LIN {X 0,Y 573.245,Z 183.073,A -85,B 0,C 180,E1 -2299.475,E2 -2299.475} C_VEL
LIN {X 0,Y 573.228,Z 183.082,A -85,B 0,C 180,E1 -2302.192,E2 -2302.192} C_VEL
LIN {X 0,Y 573.232,Z 183.075,A -85,B 0,C 180,E1 -2305.229,E2 -2305.229} C_VEL
LIN {X 0,Y 573.246,Z 183.076,A -85,B 0,C 180,E1 -2307.773,E2 -2307.773} C_VEL
LIN {X 0,Y 573.242,Z 183.077,A -85,B 0,C 180,E1 -2310.633,E2 -2310.633} C_VEL
LIN {X 0,Y 573.208,Z 183.078,A -85,B 0,C 180,E1 -2313.022,E2 -2313.022} C_VEL
LIN {X 0,Y 573.235,Z 183.076,A -85,B 0,C 180,E1 -2315.364,E2 -2315.364} C_VEL
LIN {X 0,Y 573.23,Z 183.08,A -85,B 0,C 180,E1 -2317.662,E2 -2317.662} C_VEL
LIN {X 0,Y 573.266,Z 183.072,A -85,B 0,C 180,E1 -2320.67,E2 -2320.67} C_VEL
LIN {X 0,Y 573.23,Z 183.082,A -85,B 0,C 180,E1 -2323.621,E2 -2323.621} C_VEL
LIN {X 0,Y 573.258,Z 183.081,A -85,B 0,C 180,E1 -2325.807,E2 -2325.807} C_VEL
LIN {X 0,Y 573.264,Z 183.071,A -85,B 0,C 180,E1 -2328.745,E2 -2328.745} C_VEL
LIN {X 0,Y 573.282,Z 183.078,A -85,B 0,C 180,E1 -2331.54,E2 -2331.54} C_VEL
LIN {X 0,Y 573.289,Z 183.068,A -85,B 0,C 180,E1 -2334.372,E2 -2334.372} C_VEL
LIN {X 0,Y 573.317,Z 183.067,A -85,B 0,C 180,E1 -2337.892,E2 -2337.892} C_VEL
LIN {X 0,Y 573.322,Z 183.066,A -85,B 0,C 180,E1 -2340.702,E2 -2340.702} C_VEL
LIN {X 0,Y 573.297,Z 183.071,A -85,B 0,C 180,E1 -2342.811,E2 -2342.811} C_VEL
LIN {X 0,Y 573.299,Z 183.071,A -85,B 0,C 180,E1 -2345.628,E2 -2345.628} C_VEL
LIN {X 0,Y 573.254,Z 183.074,A -85,B 0,C 180,E1 -2348.46,E2 -2348.46} C_VEL
LIN {X 0,Y 573.273,Z 183.077,A -85,B 0,C 180,E1 -2351.312,E2 -2351.312} C_VEL
LIN {X 0,Y 573.282,Z 183.073,A -85,B 0,C 180,E1 -2354.424,E2 -2354.424} C_VEL
LIN {X 0,Y 573.258,Z 183.079,A -85,B 0,C 180,E1 -2357.112,E2 -2357.112} C_VEL
LIN {X 0,Y 573.241,Z 183.076,A -85,B 0,C 180,E1 -2360.077,E2 -2360.077} C_VEL
LIN {X 0,Y 573.241,Z 183.118,A -85,B 0,C 180,E1 -2362.1,E2 -2362.1} C_VEL
LIN {X 0,Y 573.215,Z 193.051,A -85,B 0,C 180,E1 -2364.168,E2 -2364.168} C_VEL
LIN {X 0,Y 572.806,Z 194.29,A -85,B 0,C 180,E1 -2364.24,E2 -2364.24} C_VEL
LIN {X 0,Y 570.997,Z 198.736,A -85,B 0,C 180,E1 -2364.254,E2 -2364.254} C_VEL
LIN {X 0,Y 568.332,Z 207.365,A -85,B 0,C 180,E1 -2364.283,E2 -2364.283} C_VEL
LIN {X 0,Y 567.483,Z 212.853,A -85,B 0,C 180,E1 -2364.307,E2 -2364.307} C_VEL
LIN {X 0,Y 567.099,Z 223.962,A -85,B 0,C 180,E1 -2364.48,E2 -2364.48} C_VEL
LIN {X 0,Y 566.981,Z 298.738,A -85,B 0,C 180,E1 -2365.445,E2 -2365.445} C_VEL
LIN {X 0,Y 566.829,Z 311.548,A -85,B 0,C 180,E1 -2365.744,E2 -2365.744} C_VEL
LIN {X 0,Y 566.743,Z 323.735,A -85,B 0,C 180,E1 -2366.168,E2 -2366.168} C_VEL
LIN {X 0,Y 566.592,Z 335.861,A -85,B 0,C 180,E1 -2366.737,E2 -2366.737} C_VEL
LIN {X 0,Y 566.431,Z 347.166,A -85,B 0,C 180,E1 -2367.428,E2 -2367.428} C_VEL
LIN {X 0,Y 566.322,Z 357.588,A -85,B 0,C 180,E1 -2368.225,E2 -2368.225} C_VEL
LIN {X 0,Y 566.2,Z 367.478,A -85,B 0,C 180,E1 -2369.156,E2 -2369.156} C_VEL
LIN {X 0,Y 566.096,Z 376.256,A -85,B 0,C 180,E1 -2370.186,E2 -2370.186} C_VEL
LIN {X 0,Y 566.001,Z 383.39,A -85,B 0,C 180,E1 -2371.215,E2 -2371.215} C_VEL
LIN {X 0,Y 565.948,Z 389.91,A -85,B 0,C 180,E1 -2372.389,E2 -2372.389} C_VEL
LIN {X 0,Y 565.92,Z 395.392,A -85,B 0,C 180,E1 -2373.69,E2 -2373.69} C_VEL
LIN {X 0,Y 565.869,Z 399.185,A -85,B 0,C 180,E1 -2374.945,E2 -2374.945} C_VEL
LIN {X 0,Y 565.822,Z 401.595,A -85,B 0,C 180,E1 -2376.162,E2 -2376.162} C_VEL
LIN {X 0,Y 565.831,Z 402.879,A -85,B 0,C 180,E1 -2377.489,E2 -2377.489} C_VEL
LIN {X 0,Y 565.817,Z 402.903,A -85,B 0,C 180,E1 -2378.508,E2 -2378.508} C_VEL
LIN {X 0,Y 565.851,Z 401.989,A -85,B 0,C 180,E1 -2379.641,E2 -2379.641} C_VEL
LIN {X 0,Y 565.841,Z 400.12,A -85,B 0,C 180,E1 -2380.743,E2 -2380.743} C_VEL
LIN {X 0,Y 565.925,Z 396.386,A -85,B 0,C 180,E1 -2382.114,E2 -2382.114} C_VEL
LIN {X 0,Y 565.95,Z 392.76,A -85,B 0,C 180,E1 -2383.078,E2 -2383.078} C_VEL
LIN {X 0,Y 565.98,Z 386.895,A -85,B 0,C 180,E1 -2384.279,E2 -2384.279} C_VEL
LIN {X 0,Y 566.059,Z 379.21,A -85,B 0,C 180,E1 -2385.506,E2 -2385.506} C_VEL
LIN {X 0,Y 566.158,Z 371.385,A -85,B 0,C 180,E1 -2386.504,E2 -2386.504} C_VEL
LIN {X 0,Y 566.222,Z 362.446,A -85,B 0,C 180,E1 -2387.433,E2 -2387.433} C_VEL
LIN {X 0,Y 566.39,Z 352.66,A -85,B 0,C 180,E1 -2388.263,E2 -2388.263} C_VEL
LIN {X 0,Y 566.483,Z 340.994,A -85,B 0,C 180,E1 -2389.062,E2 -2389.062} C_VEL
LIN {X 0,Y 566.666,Z 329.627,A -85,B 0,C 180,E1 -2389.666,E2 -2389.666} C_VEL
LIN {X 0,Y 566.81,Z 317.931,A -85,B 0,C 180,E1 -2390.142,E2 -2390.142} C_VEL
LIN {X 0,Y 566.897,Z 304.866,A -85,B 0,C 180,E1 -2390.521,E2 -2390.521} C_VEL
LIN {X 0,Y 567.002,Z 292.327,A -85,B 0,C 180,E1 -2390.742,E2 -2390.742} C_VEL
LIN {X 0,Y 567.076,Z 198.669,A -85,B 0,C 180,E1 -2391.934,E2 -2391.934} C_VEL
LIN {X 0,Y 566.144,Z 193.381,A -85,B 0,C 180,E1 -2392.029,E2 -2392.029} C_VEL
LIN {X 0,Y 566.23,Z 183.952,A -85,B 0,C 180,E1 -2394.046,E2 -2394.046} C_VEL
LIN {X 0,Y 566.2,Z 183.956,A -85,B 0,C 180,E1 -2396.897,E2 -2396.897} C_VEL
LIN {X 0,Y 566.172,Z 183.962,A -85,B 0,C 180,E1 -2399.407,E2 -2399.407} C_VEL
LIN {X 0,Y 566.194,Z 183.953,A -85,B 0,C 180,E1 -2401.857,E2 -2401.857} C_VEL
LIN {X 0,Y 566.194,Z 183.952,A -85,B 0,C 180,E1 -2404.25,E2 -2404.25} C_VEL
LIN {X 0,Y 566.171,Z 183.959,A -85,B 0,C 180,E1 -2407.368,E2 -2407.368} C_VEL
LIN {X 0,Y 566.204,Z 183.952,A -85,B 0,C 180,E1 -2409.663,E2 -2409.663} C_VEL
LIN {X 0,Y 566.182,Z 183.953,A -85,B 0,C 180,E1 -2411.921,E2 -2411.921} C_VEL
LIN {X 0,Y 566.192,Z 183.953,A -85,B 0,C 180,E1 -2414.153,E2 -2414.153} C_VEL
LIN {X 0,Y 566.186,Z 183.956,A -85,B 0,C 180,E1 -2416.359,E2 -2416.359} C_VEL
LIN {X 0,Y 566.237,Z 183.955,A -85,B 0,C 180,E1 -2418.676,E2 -2418.676} C_VEL
LIN {X 0,Y 566.204,Z 183.951,A -85,B 0,C 180,E1 -2421.434,E2 -2421.434} C_VEL
LIN {X 0,Y 566.263,Z 183.948,A -85,B 0,C 180,E1 -2424.302,E2 -2424.302} C_VEL
LIN {X 0,Y 566.283,Z 183.942,A -85,B 0,C 180,E1 -2427.866,E2 -2427.866} C_VEL
LIN {X 0,Y 566.299,Z 183.945,A -85,B 0,C 180,E1 -2430.711,E2 -2430.711} C_VEL
LIN {X 0,Y 566.26,Z 183.947,A -85,B 0,C 180,E1 -2432.846,E2 -2432.846} C_VEL
LIN {X 0,Y 566.253,Z 183.946,A -85,B 0,C 180,E1 -2435.699,E2 -2435.699} C_VEL
LIN {X 0,Y 566.224,Z 183.954,A -85,B 0,C 180,E1 -2438.566,E2 -2438.566} C_VEL
LIN {X 0,Y 566.244,Z 183.946,A -85,B 0,C 180,E1 -2441.454,E2 -2441.454} C_VEL
LIN {X 0,Y 566.225,Z 183.952,A -85,B 0,C 180,E1 -2444.502,E2 -2444.502} C_VEL
LIN {X 0,Y 566.189,Z 183.953,A -85,B 0,C 180,E1 -2447.332,E2 -2447.332} C_VEL
LIN {X 0,Y 566.202,Z 183.954,A -85,B 0,C 180,E1 -2449.581,E2 -2449.581} C_VEL
LIN {X 0,Y 566.188,Z 183.96,A -85,B 0,C 180,E1 -2451.863,E2 -2451.863} C_VEL
LIN {X 0,Y 566.184,Z 183.953,A -85,B 0,C 180,E1 -2455.022,E2 -2455.022} C_VEL
LIN {X 0,Y 566.173,Z 183.957,A -85,B 0,C 180,E1 -2457.341,E2 -2457.341} C_VEL
LIN {X 0,Y 566.173,Z 183.964,A -85,B 0,C 180,E1 -2459.771,E2 -2459.771} C_VEL
LIN {X 0,Y 566.202,Z 183.952,A -85,B 0,C 180,E1 -2462.429,E2 -2462.429} C_VEL
LIN {X 0,Y 566.179,Z 183.955,A -85,B 0,C 180,E1 -2464.989,E2 -2464.989} C_VEL
LIN {X 0,Y 566.193,Z 183.959,A -85,B 0,C 180,E1 -2467.461,E2 -2467.461} C_VEL
LIN {X 0,Y 566.208,Z 183.951,A -85,B 0,C 180,E1 -2470.199,E2 -2470.199} C_VEL
LIN {X 0,Y 566.195,Z 183.955,A -85,B 0,C 180,E1 -2473.055,E2 -2473.055} C_VEL
LIN {X 0,Y 566.161,Z 183.957,A -85,B 0,C 180,E1 -2476.053,E2 -2476.053} C_VEL
LIN {X 0,Y 566.168,Z 183.958,A -85,B 0,C 180,E1 -2478.86,E2 -2478.86} C_VEL
LIN {X 0,Y 566.207,Z 183.957,A -85,B 0,C 180,E1 -2481.443,E2 -2481.443} C_VEL
LIN {X 0,Y 566.152,Z 183.957,A -85,B 0,C 180,E1 -2484.307,E2 -2484.307} C_VEL
LIN {X 0,Y 566.198,Z 183.957,A -85,B 0,C 180,E1 -2486.896,E2 -2486.896} C_VEL
LIN {X 0,Y 566.171,Z 183.96,A -85,B 0,C 180,E1 -2489.407,E2 -2489.407} C_VEL
LIN {X 0,Y 566.155,Z 183.957,A -85,B 0,C 180,E1 -2491.854,E2 -2491.854} C_VEL
LIN {X 0,Y 566.203,Z 183.951,A -85,B 0,C 180,E1 -2494.25,E2 -2494.25} C_VEL
LIN {X 0,Y 566.165,Z 183.958,A -85,B 0,C 180,E1 -2497.368,E2 -2497.368} C_VEL
LIN {X 0,Y 566.203,Z 183.951,A -85,B 0,C 180,E1 -2499.662,E2 -2499.662} C_VEL
LIN {X 0,Y 566.177,Z 183.954,A -85,B 0,C 180,E1 -2501.921,E2 -2501.921} C_VEL
LIN {X 0,Y 566.185,Z 183.955,A -85,B 0,C 180,E1 -2504.152,E2 -2504.152} C_VEL
LIN {X 0,Y 566.172,Z 183.959,A -85,B 0,C 180,E1 -2506.358,E2 -2506.358} C_VEL
LIN {X 0,Y 566.234,Z 183.948,A -85,B 0,C 180,E1 -2509.27,E2 -2509.27} C_VEL
LIN {X 0,Y 566.22,Z 183.952,A -85,B 0,C 180,E1 -2512.153,E2 -2512.153} C_VEL
LIN {X 0,Y 566.261,Z 183.946,A -85,B 0,C 180,E1 -2515.016,E2 -2515.016} C_VEL
LIN {X 0,Y 566.282,Z 183.943,A -85,B 0,C 180,E1 -2517.866,E2 -2517.866} C_VEL
LIN {X 0,Y 566.294,Z 183.944,A -85,B 0,C 180,E1 -2520.711,E2 -2520.711} C_VEL
LIN {X 0,Y 566.252,Z 183.947,A -85,B 0,C 180,E1 -2522.846,E2 -2522.846} C_VEL
LIN {X 0,Y 566.249,Z 183.947,A -85,B 0,C 180,E1 -2525.698,E2 -2525.698} C_VEL
LIN {X 0,Y 566.201,Z 183.955,A -85,B 0,C 180,E1 -2528.566,E2 -2528.566} C_VEL
LIN {X 0,Y 566.243,Z 183.947,A -85,B 0,C 180,E1 -2531.454,E2 -2531.454} C_VEL
LIN {X 0,Y 566.228,Z 183.95,A -85,B 0,C 180,E1 -2534.502,E2 -2534.502} C_VEL
LIN {X 0,Y 566.163,Z 183.957,A -85,B 0,C 180,E1 -2537.333,E2 -2537.333} C_VEL
LIN {X 0,Y 566.201,Z 183.956,A -85,B 0,C 180,E1 -2539.581,E2 -2539.581} C_VEL
LIN {X 0,Y 566.187,Z 183.963,A -85,B 0,C 180,E1 -2541.863,E2 -2541.863} C_VEL
LIN {X 0,Y 566.181,Z 183.954,A -85,B 0,C 180,E1 -2545.021,E2 -2545.021} C_VEL
LIN {X 0,Y 566.169,Z 183.959,A -85,B 0,C 180,E1 -2547.341,E2 -2547.341} C_VEL
LIN {X 0,Y 566.172,Z 183.963,A -85,B 0,C 180,E1 -2549.771,E2 -2549.771} C_VEL
LIN {X 0,Y 566.194,Z 183.952,A -85,B 0,C 180,E1 -2552.428,E2 -2552.428} C_VEL
LIN {X 0,Y 566.169,Z 183.957,A -85,B 0,C 180,E1 -2554.987,E2 -2554.987} C_VEL
LIN {X 0,Y 566.193,Z 183.962,A -85,B 0,C 180,E1 -2557.461,E2 -2557.461} C_VEL
LIN {X 0,Y 566.208,Z 183.951,A -85,B 0,C 180,E1 -2560.199,E2 -2560.199} C_VEL
LIN {X 0,Y 566.181,Z 183.959,A -85,B 0,C 180,E1 -2563.056,E2 -2563.056} C_VEL
LIN {X 0,Y 566.158,Z 183.957,A -85,B 0,C 180,E1 -2566.053,E2 -2566.053} C_VEL
LIN {X 0,Y 566.166,Z 183.96,A -85,B 0,C 180,E1 -2568.859,E2 -2568.859} C_VEL
LIN {X 0,Y 566.205,Z 183.955,A -85,B 0,C 180,E1 -2571.443,E2 -2571.443} C_VEL
LIN {X 0,Y 566.144,Z 183.959,A -85,B 0,C 180,E1 -2574.306,E2 -2574.306} C_VEL
LIN {X 0,Y 566.196,Z 183.96,A -85,B 0,C 180,E1 -2576.896,E2 -2576.896} C_VEL
LIN {X 0,Y 566.163,Z 183.959,A -85,B 0,C 180,E1 -2579.406,E2 -2579.406} C_VEL
LIN {X 0,Y 566.152,Z 183.959,A -85,B 0,C 180,E1 -2581.854,E2 -2581.854} C_VEL
LIN {X 0,Y 566.192,Z 183.961,A -85,B 0,C 180,E1 -2584.644,E2 -2584.644} C_VEL
LIN {X 0,Y 566.226,Z 184.037,A -85,B 0,C 180,E1 -2584.862,E2 -2584.862} C_VEL
LIN {X 0,Y 567.231,Z 189.815,A -85,B 0,C 180,E1 -2585.671,E2 -2585.671} C_VEL
LIN {X 0,Y 567.051,Z 210.5,A -85,B 0,C 180,E1 -2588.365,E2 -2588.365} C_VEL
LIN {X 0,Y 566.867,Z 231.116,A -85,B 0,C 180,E1 -2591.007,E2 -2591.007} C_VEL
LIN {X 0,Y 566.639,Z 252.903,A -85,B 0,C 180,E1 -2593.795,E2 -2593.795} C_VEL
LIN {X 0,Y 566.477,Z 270.229,A -85,B 0,C 180,E1 -2595.988,E2 -2595.988} C_VEL
LIN {X 0,Y 567.177,Z 276.49,A -85,B 0,C 180,E1 -2596.086,E2 -2596.086} C_VEL
LIN {X 0,Y 566.976,Z 378.934,A -85,B 0,C 180,E1 -2597.403,E2 -2597.403} C_VEL
LIN {X 0,Y 566.85,Z 392.21,A -85,B 0,C 180,E1 -2597.719,E2 -2597.719} C_VEL
LIN {X 0,Y 566.734,Z 404.372,A -85,B 0,C 180,E1 -2598.148,E2 -2598.148} C_VEL
LIN {X 0,Y 566.593,Z 416.405,A -85,B 0,C 180,E1 -2598.722,E2 -2598.722} C_VEL
LIN {X 0,Y 566.439,Z 428.194,A -85,B 0,C 180,E1 -2599.455,E2 -2599.455} C_VEL
LIN {X 0,Y 566.325,Z 438.601,A -85,B 0,C 180,E1 -2600.265,E2 -2600.265} C_VEL
LIN {X 0,Y 566.207,Z 447.111,A -85,B 0,C 180,E1 -2601.074,E2 -2601.074} C_VEL
LIN {X 0,Y 566.112,Z 454.959,A -85,B 0,C 180,E1 -2601.971,E2 -2601.971} C_VEL
LIN {X 0,Y 566.004,Z 462.621,A -85,B 0,C 180,E1 -2603.046,E2 -2603.046} C_VEL
LIN {X 0,Y 566.004,Z 469.679,A -85,B 0,C 180,E1 -2604.299,E2 -2604.299} C_VEL
LIN {X 0,Y 565.933,Z 474.372,A -85,B 0,C 180,E1 -2605.37,E2 -2605.37} C_VEL
LIN {X 0,Y 565.927,Z 477.957,A -85,B 0,C 180,E1 -2606.44,E2 -2606.44} C_VEL
LIN {X 0,Y 565.878,Z 479.807,A -85,B 0,C 180,E1 -2607.152,E2 -2607.152} C_VEL
LIN {X 0,Y 565.846,Z 482.184,A -85,B 0,C 180,E1 -2608.576,E2 -2608.576} C_VEL
LIN {X 0,Y 565.839,Z 483,A -85,B 0,C 180,E1 -2610,E2 -2610} C_VEL
LIN {X 0,Y 565.846,Z 482.186,A -85,B 0,C 180,E1 -2611.423,E2 -2611.423} C_VEL
LIN {X 0,Y 565.878,Z 479.81,A -85,B 0,C 180,E1 -2612.847,E2 -2612.847} C_VEL
LIN {X 0,Y 565.926,Z 476.896,A -85,B 0,C 180,E1 -2613.916,E2 -2613.916} C_VEL
LIN {X 0,Y 565.878,Z 472.949,A -85,B 0,C 180,E1 -2614.987,E2 -2614.987} C_VEL
LIN {X 0,Y 566.002,Z 467.868,A -85,B 0,C 180,E1 -2616.058,E2 -2616.058} C_VEL
LIN {X 0,Y 566.04,Z 461.469,A -85,B 0,C 180,E1 -2617.132,E2 -2617.132} C_VEL
LIN {X 0,Y 566.133,Z 453.479,A -85,B 0,C 180,E1 -2618.207,E2 -2618.207} C_VEL
LIN {X 0,Y 566.229,Z 445.336,A -85,B 0,C 180,E1 -2619.105,E2 -2619.105} C_VEL
LIN {X 0,Y 566.347,Z 435.401,A -85,B 0,C 180,E1 -2620.005,E2 -2620.005} C_VEL
LIN {X 0,Y 566.536,Z 424.294,A -85,B 0,C 180,E1 -2620.807,E2 -2620.807} C_VEL
LIN {X 0,Y 566.612,Z 413.177,A -85,B 0,C 180,E1 -2621.447,E2 -2621.447} C_VEL
LIN {X 0,Y 566.744,Z 400.984,A -85,B 0,C 180,E1 -2621.988,E2 -2621.988} C_VEL
LIN {X 0,Y 566.88,Z 388.181,A -85,B 0,C 180,E1 -2622.394,E2 -2622.394} C_VEL
LIN {X 0,Y 566.962,Z 374.612,A -85,B 0,C 180,E1 -2622.665,E2 -2622.665} C_VEL
LIN {X 0,Y 567.05,Z 274.287,A -85,B 0,C 180,E1 -2623.946,E2 -2623.946} C_VEL
LIN {X 0,Y 566.462,Z 269.947,A -85,B 0,C 180,E1 -2624.023,E2 -2624.023} C_VEL
LIN {X 0,Y 566.671,Z 247.51,A -85,B 0,C 180,E1 -2626.9,E2 -2626.9} C_VEL
LIN {X 0,Y 566.872,Z 226.532,A -85,B 0,C 180,E1 -2629.557,E2 -2629.557} C_VEL
LIN {X 0,Y 567.057,Z 205.586,A -85,B 0,C 180,E1 -2632.21,E2 -2632.21} C_VEL
LIN {X 0,Y 567.057,Z 188.967,A -85,B 0,C 180,E1 -2634.336,E2 -2634.336} C_VEL
LIN {X 0,Y 566.213,Z 183.959,A -85,B 0,C 180,E1 -2635.028,E2 -2635.028} C_VEL
LIN {X 0,Y 566.169,Z 183.963,A -85,B 0,C 180,E1 -2637.341,E2 -2637.341} C_VEL
LIN {X 0,Y 566.162,Z 183.959,A -85,B 0,C 180,E1 -2639.771,E2 -2639.771} C_VEL
LIN {X 0,Y 566.193,Z 183.955,A -85,B 0,C 180,E1 -2642.428,E2 -2642.428} C_VEL
LIN {X 0,Y 566.176,Z 183.963,A -85,B 0,C 180,E1 -2644.988,E2 -2644.988} C_VEL
LIN {X 0,Y 566.191,Z 183.954,A -85,B 0,C 180,E1 -2647.461,E2 -2647.461} C_VEL
LIN {X 0,Y 566.206,Z 183.953,A -85,B 0,C 180,E1 -2650.199,E2 -2650.199} C_VEL
LIN {X 0,Y 566.187,Z 183.957,A -85,B 0,C 180,E1 -2653.055,E2 -2653.055} C_VEL
LIN {X 0,Y 566.193,Z 183.954,A -85,B 0,C 180,E1 -2656.049,E2 -2656.049} C_VEL
LIN {X 0,Y 566.203,Z 183.951,A -85,B 0,C 180,E1 -2659.215,E2 -2659.215} C_VEL
LIN {X 0,Y 566.18,Z 183.955,A -85,B 0,C 180,E1 -2661.636,E2 -2661.636} C_VEL
LIN {X 0,Y 566.15,Z 183.967,A -85,B 0,C 180,E1 -2664.307,E2 -2664.307} C_VEL
LIN {X 0,Y 566.209,Z 183.951,A -85,B 0,C 180,E1 -2666.897,E2 -2666.897} C_VEL
LIN {X 0,Y 566.169,Z 183.956,A -85,B 0,C 180,E1 -2669.406,E2 -2669.406} C_VEL
LIN {X 0,Y 566.19,Z 183.958,A -85,B 0,C 180,E1 -2671.856,E2 -2671.856} C_VEL
LIN {X 0,Y 566.196,Z 183.959,A -85,B 0,C 180,E1 -2674.25,E2 -2674.25} C_VEL
LIN {X 0,Y 566.175,Z 183.956,A -85,B 0,C 180,E1 -2677.368,E2 -2677.368} C_VEL
LIN {X 0,Y 566.205,Z 183.956,A -85,B 0,C 180,E1 -2679.662,E2 -2679.662} C_VEL
LIN {X 0,Y 566.179,Z 183.962,A -85,B 0,C 180,E1 -2681.921,E2 -2681.921} C_VEL
LIN {X 0,Y 566.191,Z 183.952,A -85,B 0,C 180,E1 -2684.89,E2 -2684.89} C_VEL
LIN {X 0,Y 566.234,Z 183.954,A -85,B 0,C 180,E1 -2687.819,E2 -2687.819} C_VEL
LIN {X 0,Y 566.178,Z 183.958,A -85,B 0,C 180,E1 -2689.992,E2 -2689.992} C_VEL
LIN {X 0,Y 566.241,Z 183.948,A -85,B 0,C 180,E1 -2692.87,E2 -2692.87} C_VEL
LIN {X 0,Y 566.278,Z 183.945,A -85,B 0,C 180,E1 -2695.016,E2 -2695.016} C_VEL
LIN {X 0,Y 566.287,Z 183.943,A -85,B 0,C 180,E1 -2697.866,E2 -2697.866} C_VEL
LIN {X 0,Y 566.294,Z 183.941,A -85,B 0,C 180,E1 -2700.711,E2 -2700.711} C_VEL
LIN {X 0,Y 566.265,Z 183.947,A -85,B 0,C 180,E1 -2702.846,E2 -2702.846} C_VEL
LIN {X 0,Y 566.265,Z 183.946,A -85,B 0,C 180,E1 -2705.698,E2 -2705.698} C_VEL
LIN {X 0,Y 566.206,Z 183.953,A -85,B 0,C 180,E1 -2708.566,E2 -2708.566} C_VEL
LIN {X 0,Y 566.243,Z 183.951,A -85,B 0,C 180,E1 -2711.454,E2 -2711.454} C_VEL
LIN {X 0,Y 566.235,Z 183.952,A -85,B 0,C 180,E1 -2714.506,E2 -2714.506} C_VEL
LIN {X 0,Y 566.198,Z 183.956,A -85,B 0,C 180,E1 -2717.332,E2 -2717.332} C_VEL
LIN {X 0,Y 566.207,Z 183.955,A -85,B 0,C 180,E1 -2720.337,E2 -2720.337} C_VEL
LIN {X 0,Y 566.205,Z 183.982,A -85,B 0,C 180,E1 -2722.102,E2 -2722.102} C_VEL
LIN {X 0,Y 566.17,Z 193.376,A -85,B 0,C 180,E1 -2724.06,E2 -2724.06} C_VEL
LIN {X 0,Y 567.132,Z 199.084,A -85,B 0,C 180,E1 -2724.163,E2 -2724.163} C_VEL
LIN {X 0,Y 567.099,Z 223.962,A -85,B 0,C 180,E1 -2724.48,E2 -2724.48} C_VEL
LIN {X 0,Y 566.383,Z 229.808,A -85,B 0,C 180,E1 -2724.537,E2 -2724.537} C_VEL
LIN {X 0,Y 560.764,Z 248.81,A -85,B 0,C 180,E1 -2724.643,E2 -2724.643} C_VEL
LIN {X 0,Y 560.147,Z 254.652,A -85,B 0,C 180,E1 -2724.703,E2 -2724.703} C_VEL
LIN {X 0,Y 560.033,Z 299.928,A -85,B 0,C 180,E1 -2725.309,E2 -2725.309} C_VEL
LIN {X 0,Y 559.898,Z 313.312,A -85,B 0,C 180,E1 -2725.642,E2 -2725.642} C_VEL
LIN {X 0,Y 559.764,Z 326.137,A -85,B 0,C 180,E1 -2726.118,E2 -2726.118} C_VEL
LIN {X 0,Y 559.568,Z 338.61,A -85,B 0,C 180,E1 -2726.751,E2 -2726.751} C_VEL
LIN {X 0,Y 559.411,Z 349.752,A -85,B 0,C 180,E1 -2727.476,E2 -2727.476} C_VEL
LIN {X 0,Y 559.268,Z 359.399,A -85,B 0,C 180,E1 -2728.255,E2 -2728.255} C_VEL
LIN {X 0,Y 559.159,Z 368.415,A -85,B 0,C 180,E1 -2729.146,E2 -2729.146} C_VEL
LIN {X 0,Y 559.038,Z 377.03,A -85,B 0,C 180,E1 -2730.19,E2 -2730.19} C_VEL
LIN {X 0,Y 558.923,Z 384.053,A -85,B 0,C 180,E1 -2731.236,E2 -2731.236} C_VEL
LIN {X 0,Y 558.89,Z 389.486,A -85,B 0,C 180,E1 -2732.233,E2 -2732.233} C_VEL
LIN {X 0,Y 558.824,Z 395.266,A -85,B 0,C 180,E1 -2733.598,E2 -2733.598} C_VEL
LIN {X 0,Y 558.8,Z 398.048,A -85,B 0,C 180,E1 -2734.469,E2 -2734.469} C_VEL
LIN {X 0,Y 558.756,Z 400.199,A -85,B 0,C 180,E1 -2735.351,E2 -2735.351} C_VEL
LIN {X 0,Y 558.733,Z 401.945,A -85,B 0,C 180,E1 -2736.388,E2 -2736.388} C_VEL
LIN {X 0,Y 558.741,Z 402.905,A -85,B 0,C 180,E1 -2737.587,E2 -2737.587} C_VEL
LIN {X 0,Y 558.73,Z 402.649,A -85,B 0,C 180,E1 -2738.971,E2 -2738.971} C_VEL
LIN {X 0,Y 558.764,Z 401.671,A -85,B 0,C 180,E1 -2739.901,E2 -2739.901} C_VEL
LIN {X 0,Y 558.758,Z 399.63,A -85,B 0,C 180,E1 -2741.003,E2 -2741.003} C_VEL
LIN {X 0,Y 558.835,Z 395.546,A -85,B 0,C 180,E1 -2742.411,E2 -2742.411} C_VEL
LIN {X 0,Y 558.848,Z 391.448,A -85,B 0,C 180,E1 -2743.439,E2 -2743.439} C_VEL
LIN {X 0,Y 558.916,Z 386.331,A -85,B 0,C 180,E1 -2744.46,E2 -2744.46} C_VEL
LIN {X 0,Y 559.01,Z 378.632,A -85,B 0,C 180,E1 -2745.684,E2 -2745.684} C_VEL
LIN {X 0,Y 559.135,Z 369.656,A -85,B 0,C 180,E1 -2746.805,E2 -2746.805} C_VEL
LIN {X 0,Y 559.273,Z 360.305,A -85,B 0,C 180,E1 -2747.751,E2 -2747.751} C_VEL
LIN {X 0,Y 559.398,Z 349.744,A -85,B 0,C 180,E1 -2748.614,E2 -2748.614} C_VEL
LIN {X 0,Y 559.554,Z 338.856,A -85,B 0,C 180,E1 -2749.325,E2 -2749.325} C_VEL
LIN {X 0,Y 559.772,Z 326.579,A -85,B 0,C 180,E1 -2749.952,E2 -2749.952} C_VEL
LIN {X 0,Y 559.898,Z 313.913,A -85,B 0,C 180,E1 -2750.43,E2 -2750.43} C_VEL
LIN {X 0,Y 559.99,Z 301.114,A -85,B 0,C 180,E1 -2750.758,E2 -2750.758} C_VEL
LIN {X 0,Y 560.078,Z 277.814,A -85,B 0,C 180,E1 -2751.089,E2 -2751.089} C_VEL
LIN {X 0,Y 560.219,Z 199.597,A -85,B 0,C 180,E1 -2752.097,E2 -2752.097} C_VEL
LIN {X 0,Y 559.137,Z 193.6,A -85,B 0,C 180,E1 -2752.215,E2 -2752.215} C_VEL
LIN {X 0,Y 559.186,Z 184.829,A -85,B 0,C 180,E1 -2754.071,E2 -2754.071} C_VEL
LIN {X 0,Y 559.151,Z 184.839,A -85,B 0,C 180,E1 -2757.285,E2 -2757.285} C_VEL
LIN {X 0,Y 559.143,Z 184.83,A -85,B 0,C 180,E1 -2760.144,E2 -2760.144} C_VEL
LIN {X 0,Y 559.16,Z 184.837,A -85,B 0,C 180,E1 -2763.097,E2 -2763.097} C_VEL
LIN {X 0,Y 559.124,Z 184.836,A -85,B 0,C 180,E1 -2765.494,E2 -2765.494} C_VEL
LIN {X 0,Y 559.172,Z 184.83,A -85,B 0,C 180,E1 -2768.624,E2 -2768.624} C_VEL
LIN {X 0,Y 559.16,Z 184.838,A -85,B 0,C 180,E1 -2770.926,E2 -2770.926} C_VEL
LIN {X 0,Y 559.155,Z 184.829,A -85,B 0,C 180,E1 -2773.948,E2 -2773.948} C_VEL
LIN {X 0,Y 559.16,Z 184.829,A -85,B 0,C 180,E1 -2776.184,E2 -2776.184} C_VEL
LIN {X 0,Y 559.193,Z 184.828,A -85,B 0,C 180,E1 -2779.134,E2 -2779.134} C_VEL
LIN {X 0,Y 559.196,Z 184.825,A -85,B 0,C 180,E1 -2782.054,E2 -2782.054} C_VEL
LIN {X 0,Y 559.246,Z 184.822,A -85,B 0,C 180,E1 -2784.953,E2 -2784.953} C_VEL
LIN {X 0,Y 559.253,Z 184.817,A -85,B 0,C 180,E1 -2787.84,E2 -2787.84} C_VEL
LIN {X 0,Y 559.27,Z 184.82,A -85,B 0,C 180,E1 -2790.72,E2 -2790.72} C_VEL
LIN {X 0,Y 559.226,Z 184.823,A -85,B 0,C 180,E1 -2792.882,E2 -2792.882} C_VEL
LIN {X 0,Y 559.223,Z 184.822,A -85,B 0,C 180,E1 -2795.77,E2 -2795.77} C_VEL
LIN {X 0,Y 559.183,Z 184.829,A -85,B 0,C 180,E1 -2798.675,E2 -2798.675} C_VEL
LIN {X 0,Y 559.207,Z 184.824,A -85,B 0,C 180,E1 -2801.601,E2 -2801.601} C_VEL
LIN {X 0,Y 559.183,Z 184.828,A -85,B 0,C 180,E1 -2804.588,E2 -2804.588} C_VEL
LIN {X 0,Y 559.134,Z 184.834,A -85,B 0,C 180,E1 -2807.558,E2 -2807.558} C_VEL
LIN {X 0,Y 559.166,Z 184.834,A -85,B 0,C 180,E1 -2809.838,E2 -2809.838} C_VEL
LIN {X 0,Y 559.136,Z 184.838,A -85,B 0,C 180,E1 -2812.153,E2 -2812.153} C_VEL
LIN {X 0,Y 559.143,Z 184.831,A -85,B 0,C 180,E1 -2815.179,E2 -2815.179} C_VEL
LIN {X 0,Y 559.129,Z 184.84,A -85,B 0,C 180,E1 -2817.715,E2 -2817.715} C_VEL
LIN {X 0,Y 559.139,Z 184.834,A -85,B 0,C 180,E1 -2820.184,E2 -2820.184} C_VEL
LIN {X 0,Y 559.155,Z 184.829,A -85,B 0,C 180,E1 -2822.716,E2 -2822.716} C_VEL
LIN {X 0,Y 559.124,Z 184.837,A -85,B 0,C 180,E1 -2825.325,E2 -2825.325} C_VEL
LIN {X 0,Y 559.13,Z 184.835,A -85,B 0,C 180,E1 -2828.018,E2 -2828.018} C_VEL
LIN {X 0,Y 559.157,Z 184.829,A -85,B 0,C 180,E1 -2830.813,E2 -2830.813} C_VEL
LIN {X 0,Y 559.138,Z 184.836,A -85,B 0,C 180,E1 -2833.735,E2 -2833.735} C_VEL
LIN {X 0,Y 559.133,Z 184.833,A -85,B 0,C 180,E1 -2836.805,E2 -2836.805} C_VEL
LIN {X 0,Y 559.155,Z 184.836,A -85,B 0,C 180,E1 -2839.187,E2 -2839.187} C_VEL
LIN {X 0,Y 559.13,Z 184.833,A -85,B 0,C 180,E1 -2841.982,E2 -2841.982} C_VEL
LIN {X 0,Y 559.131,Z 184.835,A -85,B 0,C 180,E1 -2844.788,E2 -2844.788} C_VEL
LIN {X 0,Y 559.151,Z 184.835,A -85,B 0,C 180,E1 -2847.366,E2 -2847.366} C_VEL
LIN {X 0,Y 559.121,Z 184.833,A -85,B 0,C 180,E1 -2850.148,E2 -2850.148} C_VEL
LIN {X 0,Y 559.166,Z 184.834,A -85,B 0,C 180,E1 -2853.174,E2 -2853.174} C_VEL
LIN {X 0,Y 559.118,Z 184.835,A -85,B 0,C 180,E1 -2855.493,E2 -2855.493} C_VEL
LIN {X 0,Y 559.174,Z 184.832,A -85,B 0,C 180,E1 -2858.624,E2 -2858.624} C_VEL
LIN {X 0,Y 559.159,Z 184.836,A -85,B 0,C 180,E1 -2860.926,E2 -2860.926} C_VEL
LIN {X 0,Y 559.145,Z 184.83,A -85,B 0,C 180,E1 -2863.947,E2 -2863.947} C_VEL
LIN {X 0,Y 559.149,Z 184.832,A -85,B 0,C 180,E1 -2866.184,E2 -2866.184} C_VEL
LIN {X 0,Y 559.193,Z 184.826,A -85,B 0,C 180,E1 -2869.134,E2 -2869.134} C_VEL
LIN {X 0,Y 559.191,Z 184.827,A -85,B 0,C 180,E1 -2872.053,E2 -2872.053} C_VEL
LIN {X 0,Y 559.238,Z 184.821,A -85,B 0,C 180,E1 -2874.953,E2 -2874.953} C_VEL
LIN {X 0,Y 559.253,Z 184.818,A -85,B 0,C 180,E1 -2877.839,E2 -2877.839} C_VEL
LIN {X 0,Y 559.265,Z 184.819,A -85,B 0,C 180,E1 -2880.72,E2 -2880.72} C_VEL
LIN {X 0,Y 559.219,Z 184.822,A -85,B 0,C 180,E1 -2882.882,E2 -2882.882} C_VEL
LIN {X 0,Y 559.218,Z 184.824,A -85,B 0,C 180,E1 -2885.77,E2 -2885.77} C_VEL
LIN {X 0,Y 559.165,Z 184.83,A -85,B 0,C 180,E1 -2888.675,E2 -2888.675} C_VEL
LIN {X 0,Y 559.204,Z 184.825,A -85,B 0,C 180,E1 -2891.601,E2 -2891.601} C_VEL
LIN {X 0,Y 559.185,Z 184.827,A -85,B 0,C 180,E1 -2894.588,E2 -2894.588} C_VEL
LIN {X 0,Y 559.118,Z 184.837,A -85,B 0,C 180,E1 -2897.558,E2 -2897.558} C_VEL
LIN {X 0,Y 559.163,Z 184.837,A -85,B 0,C 180,E1 -2899.838,E2 -2899.838} C_VEL
LIN {X 0,Y 559.133,Z 184.836,A -85,B 0,C 180,E1 -2902.153,E2 -2902.153} C_VEL
LIN {X 0,Y 559.142,Z 184.832,A -85,B 0,C 180,E1 -2905.178,E2 -2905.178} C_VEL
LIN {X 0,Y 559.111,Z 184.844,A -85,B 0,C 180,E1 -2907.716,E2 -2907.716} C_VEL
LIN {X 0,Y 559.138,Z 184.833,A -85,B 0,C 180,E1 -2910.184,E2 -2910.184} C_VEL
LIN {X 0,Y 559.15,Z 184.829,A -85,B 0,C 180,E1 -2912.716,E2 -2912.716} C_VEL
LIN {X 0,Y 559.119,Z 184.84,A -85,B 0,C 180,E1 -2915.325,E2 -2915.325} C_VEL
LIN {X 0,Y 559.129,Z 184.834,A -85,B 0,C 180,E1 -2918.018,E2 -2918.018} C_VEL
LIN {X 0,Y 559.155,Z 184.83,A -85,B 0,C 180,E1 -2920.813,E2 -2920.813} C_VEL
LIN {X 0,Y 559.11,Z 184.838,A -85,B 0,C 180,E1 -2923.737,E2 -2923.737} C_VEL
LIN {X 0,Y 559.109,Z 184.834,A -85,B 0,C 180,E1 -2926.263,E2 -2926.263} C_VEL
LIN {X 0,Y 559.155,Z 184.839,A -85,B 0,C 180,E1 -2929.187,E2 -2929.187} C_VEL
LIN {X 0,Y 559.129,Z 184.832,A -85,B 0,C 180,E1 -2931.982,E2 -2931.982} C_VEL
LIN {X 0,Y 559.125,Z 184.838,A -85,B 0,C 180,E1 -2934.789,E2 -2934.789} C_VEL
LIN {X 0,Y 559.151,Z 184.834,A -85,B 0,C 180,E1 -2937.366,E2 -2937.366} C_VEL
LIN {X 0,Y 559.113,Z 184.835,A -85,B 0,C 180,E1 -2940.15,E2 -2940.15} C_VEL
LIN {X 0,Y 559.128,Z 184.839,A -85,B 0,C 180,E1 -2943.182,E2 -2943.182} C_VEL
LIN {X 0,Y 559.17,Z 184.941,A -85,B 0,C 180,E1 -2944.701,E2 -2944.701} C_VEL
LIN {X 0,Y 560.364,Z 192.347,A -85,B 0,C 180,E1 -2945.748,E2 -2945.748} C_VEL
LIN {X 0,Y 560.055,Z 212.755,A -85,B 0,C 180,E1 -2948.436,E2 -2948.436} C_VEL
LIN {X 0,Y 559.864,Z 233.612,A -85,B 0,C 180,E1 -2951.141,E2 -2951.141} C_VEL
LIN {X 0,Y 559.565,Z 257.084,A -85,B 0,C 180,E1 -2954.146,E2 -2954.146} C_VEL
LIN {X 0,Y 559.469,Z 270.229,A -85,B 0,C 180,E1 -2955.809,E2 -2955.809} C_VEL
LIN {X 0,Y 560.303,Z 277.11,A -85,B 0,C 180,E1 -2955.92,E2 -2955.92} C_VEL
LIN {X 0,Y 560.068,Z 378.934,A -85,B 0,C 180,E1 -2957.245,E2 -2957.245} C_VEL
LIN {X 0,Y 559.917,Z 392.209,A -85,B 0,C 180,E1 -2957.564,E2 -2957.564} C_VEL
LIN {X 0,Y 559.769,Z 405.491,A -85,B 0,C 180,E1 -2958.044,E2 -2958.044} C_VEL
LIN {X 0,Y 559.605,Z 417.418,A -85,B 0,C 180,E1 -2958.638,E2 -2958.638} C_VEL
LIN {X 0,Y 559.426,Z 429.483,A -85,B 0,C 180,E1 -2959.413,E2 -2959.413} C_VEL
LIN {X 0,Y 559.297,Z 439.644,A -85,B 0,C 180,E1 -2960.233,E2 -2960.233} C_VEL
LIN {X 0,Y 559.134,Z 448.784,A -85,B 0,C 180,E1 -2961.142,E2 -2961.142} C_VEL
LIN {X 0,Y 559.01,Z 457.687,A -85,B 0,C 180,E1 -2962.232,E2 -2962.232} C_VEL
LIN {X 0,Y 558.925,Z 463.738,A -85,B 0,C 180,E1 -2963.14,E2 -2963.14} C_VEL
LIN {X 0,Y 558.936,Z 469.678,A -85,B 0,C 180,E1 -2964.227,E2 -2964.227} C_VEL
LIN {X 0,Y 558.826,Z 474.372,A -85,B 0,C 180,E1 -2965.311,E2 -2965.311} C_VEL
LIN {X 0,Y 558.836,Z 477.958,A -85,B 0,C 180,E1 -2966.395,E2 -2966.395} C_VEL
LIN {X 0,Y 558.799,Z 479.807,A -85,B 0,C 180,E1 -2967.116,E2 -2967.116} C_VEL
LIN {X 0,Y 558.745,Z 482.183,A -85,B 0,C 180,E1 -2968.558,E2 -2968.558} C_VEL
LIN {X 0,Y 558.74,Z 483,A -85,B 0,C 180,E1 -2970,E2 -2970} C_VEL
LIN {X 0,Y 558.745,Z 482.185,A -85,B 0,C 180,E1 -2971.441,E2 -2971.441} C_VEL
LIN {X 0,Y 558.799,Z 479.81,A -85,B 0,C 180,E1 -2972.883,E2 -2972.883} C_VEL
LIN {X 0,Y 558.844,Z 476.896,A -85,B 0,C 180,E1 -2973.966,E2 -2973.966} C_VEL
LIN {X 0,Y 558.798,Z 472.949,A -85,B 0,C 180,E1 -2975.051,E2 -2975.051} C_VEL
LIN {X 0,Y 558.919,Z 467.868,A -85,B 0,C 180,E1 -2976.135,E2 -2976.135} C_VEL
LIN {X 0,Y 558.977,Z 461.468,A -85,B 0,C 180,E1 -2977.223,E2 -2977.223} C_VEL
LIN {X 0,Y 559.099,Z 453.479,A -85,B 0,C 180,E1 -2978.311,E2 -2978.311} C_VEL
LIN {X 0,Y 559.194,Z 445.335,A -85,B 0,C 180,E1 -2979.221,E2 -2979.221} C_VEL
LIN {X 0,Y 559.357,Z 435.4,A -85,B 0,C 180,E1 -2980.131,E2 -2980.131} C_VEL
LIN {X 0,Y 559.556,Z 424.4,A -85,B 0,C 180,E1 -2980.936,E2 -2980.936} C_VEL
LIN {X 0,Y 559.671,Z 412.461,A -85,B 0,C 180,E1 -2981.628,E2 -2981.628} C_VEL
LIN {X 0,Y 559.796,Z 400.982,A -85,B 0,C 180,E1 -2982.139,E2 -2982.139} C_VEL
LIN {X 0,Y 559.944,Z 388.18,A -85,B 0,C 180,E1 -2982.55,E2 -2982.55} C_VEL
LIN {X 0,Y 560.062,Z 374.611,A -85,B 0,C 180,E1 -2982.824,E2 -2982.824} C_VEL
LIN {X 0,Y 560.145,Z 274.732,A -85,B 0,C 180,E1 -2984.115,E2 -2984.115} C_VEL
LIN {X 0,Y 559.471,Z 269.947,A -85,B 0,C 180,E1 -2984.202,E2 -2984.202} C_VEL
LIN {X 0,Y 559.675,Z 245.771,A -85,B 0,C 180,E1 -2987.278,E2 -2987.278} C_VEL
LIN {X 0,Y 559.882,Z 224.347,A -85,B 0,C 180,E1 -2990.002,E2 -2990.002} C_VEL
LIN {X 0,Y 560.101,Z 201.88,A -85,B 0,C 180,E1 -2992.891,E2 -2992.891} C_VEL
LIN {X 0,Y 560.03,Z 189.705,A -85,B 0,C 180,E1 -2994.464,E2 -2994.464} C_VEL
LIN {X 0,Y 559.16,Z 184.838,A -85,B 0,C 180,E1 -2995.134,E2 -2995.134} C_VEL
LIN {X 0,Y 559.11,Z 184.838,A -85,B 0,C 180,E1 -2997.716,E2 -2997.716} C_VEL
LIN {X 0,Y 559.13,Z 184.834,A -85,B 0,C 180,E1 -3000.184,E2 -3000.184} C_VEL
LIN {X 0,Y 559.148,Z 184.837,A -85,B 0,C 180,E1 -3002.716,E2 -3002.716} C_VEL
LIN {X 0,Y 559.122,Z 184.836,A -85,B 0,C 180,E1 -3005.324,E2 -3005.324} C_VEL
LIN {X 0,Y 559.127,Z 184.833,A -85,B 0,C 180,E1 -3008.018,E2 -3008.018} C_VEL
LIN {X 0,Y 559.154,Z 184.837,A -85,B 0,C 180,E1 -3010.812,E2 -3010.812} C_VEL
LIN {X 0,Y 559.11,Z 184.835,A -85,B 0,C 180,E1 -3013.737,E2 -3013.737} C_VEL
LIN {X 0,Y 559.136,Z 184.836,A -85,B 0,C 180,E1 -3016.265,E2 -3016.265} C_VEL
LIN {X 0,Y 559.155,Z 184.83,A -85,B 0,C 180,E1 -3019.187,E2 -3019.187} C_VEL
LIN {X 0,Y 559.128,Z 184.836,A -85,B 0,C 180,E1 -3021.982,E2 -3021.982} C_VEL
LIN {X 0,Y 559.128,Z 184.835,A -85,B 0,C 180,E1 -3024.788,E2 -3024.788} C_VEL
LIN {X 0,Y 559.153,Z 184.829,A -85,B 0,C 180,E1 -3027.365,E2 -3027.365} C_VEL
LIN {X 0,Y 559.138,Z 184.84,A -85,B 0,C 180,E1 -3030.144,E2 -3030.144} C_VEL
LIN {X 0,Y 559.159,Z 184.828,A -85,B 0,C 180,E1 -3033.175,E2 -3033.175} C_VEL
LIN {X 0,Y 559.125,Z 184.835,A -85,B 0,C 180,E1 -3035.493,E2 -3035.493} C_VEL
LIN {X 0,Y 559.172,Z 184.828,A -85,B 0,C 180,E1 -3038.624,E2 -3038.624} C_VEL
LIN {X 0,Y 559.158,Z 184.829,A -85,B 0,C 180,E1 -3040.926,E2 -3040.926} C_VEL
LIN {X 0,Y 559.146,Z 184.837,A -85,B 0,C 180,E1 -3043.947,E2 -3043.947} C_VEL
LIN {X 0,Y 559.161,Z 184.831,A -85,B 0,C 180,E1 -3046.184,E2 -3046.184} C_VEL
LIN {X 0,Y 559.195,Z 184.826,A -85,B 0,C 180,E1 -3049.133,E2 -3049.133} C_VEL
LIN {X 0,Y 559.199,Z 184.827,A -85,B 0,C 180,E1 -3052.053,E2 -3052.053} C_VEL
LIN {X 0,Y 559.252,Z 184.819,A -85,B 0,C 180,E1 -3054.953,E2 -3054.953} C_VEL
LIN {X 0,Y 559.257,Z 184.819,A -85,B 0,C 180,E1 -3057.839,E2 -3057.839} C_VEL
LIN {X 0,Y 559.266,Z 184.817,A -85,B 0,C 180,E1 -3060.72,E2 -3060.72} C_VEL
LIN {X 0,Y 559.233,Z 184.824,A -85,B 0,C 180,E1 -3062.881,E2 -3062.881} C_VEL
LIN {X 0,Y 559.233,Z 184.821,A -85,B 0,C 180,E1 -3065.77,E2 -3065.77} C_VEL
LIN {X 0,Y 559.17,Z 184.831,A -85,B 0,C 180,E1 -3068.675,E2 -3068.675} C_VEL
LIN {X 0,Y 559.206,Z 184.826,A -85,B 0,C 180,E1 -3071.6,E2 -3071.6} C_VEL
LIN {X 0,Y 559.201,Z 184.829,A -85,B 0,C 180,E1 -3074.595,E2 -3074.595} C_VEL
LIN {X 0,Y 559.141,Z 184.833,A -85,B 0,C 180,E1 -3077.557,E2 -3077.557} C_VEL
LIN {X 0,Y 559.166,Z 184.829,A -85,B 0,C 180,E1 -3079.838,E2 -3079.838} C_VEL
LIN {X 0,Y 559.174,Z 184.99,A -85,B 0,C 180,E1 -3082.151,E2 -3082.151} C_VEL
LIN {X 0,Y 559.138,Z 193.38,A -85,B 0,C 180,E1 -3083.865,E2 -3083.865} C_VEL
LIN {X 0,Y 560.274,Z 200.809,A -85,B 0,C 180,E1 -3084.01,E2 -3084.01} C_VEL
LIN {X 0,Y 560.147,Z 254.652,A -85,B 0,C 180,E1 -3084.703,E2 -3084.703} C_VEL
LIN {X 0,Y 559.517,Z 260.498,A -85,B 0,C 180,E1 -3084.763,E2 -3084.763} C_VEL
LIN {X 0,Y 553.852,Z 279.498,A -85,B 0,C 180,E1 -3084.87,E2 -3084.87} C_VEL
LIN {X 0,Y 553.192,Z 285.344,A -85,B 0,C 180,E1 -3084.932,E2 -3084.932} C_VEL
LIN {X 0,Y 553.082,Z 302.463,A -85,B 0,C 180,E1 -3085.194,E2 -3085.194} C_VEL
LIN {X 0,Y 552.99,Z 315.167,A -85,B 0,C 180,E1 -3085.532,E2 -3085.532} C_VEL
LIN {X 0,Y 552.807,Z 327.548,A -85,B 0,C 180,E1 -3086.015,E2 -3086.015} C_VEL
LIN {X 0,Y 552.605,Z 339.16,A -85,B 0,C 180,E1 -3086.62,E2 -3086.62} C_VEL
LIN {X 0,Y 552.421,Z 350.292,A -85,B 0,C 180,E1 -3087.361,E2 -3087.361} C_VEL
LIN {X 0,Y 552.271,Z 359.152,A -85,B 0,C 180,E1 -3088.089,E2 -3088.089} C_VEL
LIN {X 0,Y 552.138,Z 367.608,A -85,B 0,C 180,E1 -3088.927,E2 -3088.927} C_VEL
LIN {X 0,Y 551.996,Z 376.639,A -85,B 0,C 180,E1 -3090.029,E2 -3090.029} C_VEL
LIN {X 0,Y 551.858,Z 384.537,A -85,B 0,C 180,E1 -3091.228,E2 -3091.228} C_VEL
LIN {X 0,Y 551.786,Z 390.378,A -85,B 0,C 180,E1 -3092.34,E2 -3092.34} C_VEL
LIN {X 0,Y 551.747,Z 395.63,A -85,B 0,C 180,E1 -3093.648,E2 -3093.648} C_VEL
LIN {X 0,Y 551.677,Z 399.463,A -85,B 0,C 180,E1 -3094.979,E2 -3094.979} C_VEL
LIN {X 0,Y 551.64,Z 401.231,A -85,B 0,C 180,E1 -3095.877,E2 -3095.877} C_VEL
LIN {X 0,Y 551.645,Z 402.4,A -85,B 0,C 180,E1 -3096.783,E2 -3096.783} C_VEL
LIN {X 0,Y 551.63,Z 402.958,A -85,B 0,C 180,E1 -3097.823,E2 -3097.823} C_VEL
LIN {X 0,Y 551.64,Z 402.637,A -85,B 0,C 180,E1 -3099,E2 -3099} C_VEL
LIN {X 0,Y 551.65,Z 401.329,A -85,B 0,C 180,E1 -3100.147,E2 -3100.147} C_VEL
LIN {X 0,Y 551.719,Z 398.552,A -85,B 0,C 180,E1 -3101.483,E2 -3101.483} C_VEL
LIN {X 0,Y 551.749,Z 395.563,A -85,B 0,C 180,E1 -3102.462,E2 -3102.462} C_VEL
LIN {X 0,Y 551.765,Z 390.563,A -85,B 0,C 180,E1 -3103.709,E2 -3103.709} C_VEL
LIN {X 0,Y 551.85,Z 383.848,A -85,B 0,C 180,E1 -3104.976,E2 -3104.976} C_VEL
LIN {X 0,Y 551.981,Z 376.642,A -85,B 0,C 180,E1 -3106.06,E2 -3106.06} C_VEL
LIN {X 0,Y 552.119,Z 368.362,A -85,B 0,C 180,E1 -3107.078,E2 -3107.078} C_VEL
LIN {X 0,Y 552.282,Z 359.6,A -85,B 0,C 180,E1 -3107.958,E2 -3107.958} C_VEL
LIN {X 0,Y 552.419,Z 350.457,A -85,B 0,C 180,E1 -3108.715,E2 -3108.715} C_VEL
LIN {X 0,Y 552.602,Z 339.578,A -85,B 0,C 180,E1 -3109.443,E2 -3109.443} C_VEL
LIN {X 0,Y 552.817,Z 327.856,A -85,B 0,C 180,E1 -3110.058,E2 -3110.058} C_VEL
LIN {X 0,Y 552.976,Z 315.531,A -85,B 0,C 180,E1 -3110.545,E2 -3110.545} C_VEL
LIN {X 0,Y 553.082,Z 302.523,A -85,B 0,C 180,E1 -3110.894,E2 -3110.894} C_VEL
LIN {X 0,Y 553.191,Z 282.197,A -85,B 0,C 180,E1 -3111.2,E2 -3111.2} C_VEL
LIN {X 0,Y 553.316,Z 200.298,A -85,B 0,C 180,E1 -3112.269,E2 -3112.269} C_VEL
LIN {X 0,Y 552.152,Z 193.89,A -85,B 0,C 180,E1 -3112.399,E2 -3112.399} C_VEL
LIN {X 0,Y 552.15,Z 185.706,A -85,B 0,C 180,E1 -3114.105,E2 -3114.105} C_VEL
LIN {X 0,Y 552.11,Z 185.715,A -85,B 0,C 180,E1 -3117.155,E2 -3117.155} C_VEL
LIN {X 0,Y 552.112,Z 185.707,A -85,B 0,C 180,E1 -3119.951,E2 -3119.951} C_VEL
LIN {X 0,Y 552.131,Z 185.711,A -85,B 0,C 180,E1 -3123.002,E2 -3123.002} C_VEL
LIN {X 0,Y 552.085,Z 185.71,A -85,B 0,C 180,E1 -3125.961,E2 -3125.961} C_VEL
LIN {X 0,Y 552.118,Z 185.713,A -85,B 0,C 180,E1 -3129.12,E2 -3129.12} C_VEL
LIN {X 0,Y 552.089,Z 185.711,A -85,B 0,C 180,E1 -3131.443,E2 -3131.443} C_VEL
LIN {X 0,Y 552.105,Z 185.707,A -85,B 0,C 180,E1 -3133.737,E2 -3133.737} C_VEL
LIN {X 0,Y 552.123,Z 185.705,A -85,B 0,C 180,E1 -3136.004,E2 -3136.004} C_VEL
LIN {X 0,Y 552.162,Z 185.706,A -85,B 0,C 180,E1 -3138.994,E2 -3138.994} C_VEL
LIN {X 0,Y 552.15,Z 185.702,A -85,B 0,C 180,E1 -3141.952,E2 -3141.952} C_VEL
LIN {X 0,Y 552.222,Z 185.698,A -85,B 0,C 180,E1 -3144.889,E2 -3144.889} C_VEL
LIN {X 0,Y 552.225,Z 185.693,A -85,B 0,C 180,E1 -3147.812,E2 -3147.812} C_VEL
LIN {X 0,Y 552.24,Z 185.696,A -85,B 0,C 180,E1 -3150.729,E2 -3150.729} C_VEL
LIN {X 0,Y 552.192,Z 185.699,A -85,B 0,C 180,E1 -3152.918,E2 -3152.918} C_VEL
LIN {X 0,Y 552.193,Z 185.698,A -85,B 0,C 180,E1 -3155.844,E2 -3155.844} C_VEL
LIN {X 0,Y 552.151,Z 185.704,A -85,B 0,C 180,E1 -3158.786,E2 -3158.786} C_VEL
LIN {X 0,Y 552.163,Z 185.702,A -85,B 0,C 180,E1 -3161.751,E2 -3161.751} C_VEL
LIN {X 0,Y 552.131,Z 185.705,A -85,B 0,C 180,E1 -3164.749,E2 -3164.749} C_VEL
LIN {X 0,Y 552.092,Z 185.714,A -85,B 0,C 180,E1 -3167.789,E2 -3167.789} C_VEL
LIN {X 0,Y 552.127,Z 185.713,A -85,B 0,C 180,E1 -3170.102,E2 -3170.102} C_VEL
LIN {X 0,Y 552.088,Z 185.712,A -85,B 0,C 180,E1 -3172.451,E2 -3172.451} C_VEL
LIN {X 0,Y 552.088,Z 185.711,A -85,B 0,C 180,E1 -3175.335,E2 -3175.335} C_VEL
LIN {X 0,Y 552.079,Z 185.716,A -85,B 0,C 180,E1 -3178.1,E2 -3178.1} C_VEL
LIN {X 0,Y 552.095,Z 185.708,A -85,B 0,C 180,E1 -3180.61,E2 -3180.61} C_VEL
LIN {X 0,Y 552.115,Z 185.708,A -85,B 0,C 180,E1 -3183.186,E2 -3183.186} C_VEL
LIN {X 0,Y 552.076,Z 185.717,A -85,B 0,C 180,E1 -3185.845,E2 -3185.845} C_VEL
LIN {X 0,Y 552.116,Z 185.706,A -85,B 0,C 180,E1 -3188.589,E2 -3188.589} C_VEL
LIN {X 0,Y 552.113,Z 185.715,A -85,B 0,C 180,E1 -3191.447,E2 -3191.447} C_VEL
LIN {X 0,Y 552.09,Z 185.709,A -85,B 0,C 180,E1 -3194.531,E2 -3194.531} C_VEL
LIN {X 0,Y 552.111,Z 185.712,A -85,B 0,C 180,E1 -3197.587,E2 -3197.587} C_VEL
LIN {X 0,Y 552.129,Z 185.704,A -85,B 0,C 180,E1 -3200.473,E2 -3200.473} C_VEL
LIN {X 0,Y 552.101,Z 185.716,A -85,B 0,C 180,E1 -3203.318,E2 -3203.318} C_VEL
LIN {X 0,Y 552.103,Z 185.708,A -85,B 0,C 180,E1 -3205.937,E2 -3205.937} C_VEL
LIN {X 0,Y 552.123,Z 185.707,A -85,B 0,C 180,E1 -3208.541,E2 -3208.541} C_VEL
LIN {X 0,Y 552.083,Z 185.713,A -85,B 0,C 180,E1 -3211.447,E2 -3211.447} C_VEL
LIN {X 0,Y 552.113,Z 185.708,A -85,B 0,C 180,E1 -3213.543,E2 -3213.543} C_VEL
LIN {X 0,Y 552.091,Z 185.716,A -85,B 0,C 180,E1 -3216.758,E2 -3216.758} C_VEL
LIN {X 0,Y 552.118,Z 185.711,A -85,B 0,C 180,E1 -3219.12,E2 -3219.12} C_VEL
LIN {X 0,Y 552.086,Z 185.711,A -85,B 0,C 180,E1 -3221.443,E2 -3221.443} C_VEL
LIN {X 0,Y 552.094,Z 185.708,A -85,B 0,C 180,E1 -3223.737,E2 -3223.737} C_VEL
LIN {X 0,Y 552.116,Z 185.707,A -85,B 0,C 180,E1 -3226.004,E2 -3226.004} C_VEL
LIN {X 0,Y 552.162,Z 185.704,A -85,B 0,C 180,E1 -3228.993,E2 -3228.993} C_VEL
LIN {X 0,Y 552.147,Z 185.703,A -85,B 0,C 180,E1 -3231.951,E2 -3231.951} C_VEL
LIN {X 0,Y 552.214,Z 185.697,A -85,B 0,C 180,E1 -3234.889,E2 -3234.889} C_VEL
LIN {X 0,Y 552.224,Z 185.694,A -85,B 0,C 180,E1 -3237.812,E2 -3237.812} C_VEL
LIN {X 0,Y 552.236,Z 185.694,A -85,B 0,C 180,E1 -3240.729,E2 -3240.729} C_VEL
LIN {X 0,Y 552.186,Z 185.698,A -85,B 0,C 180,E1 -3242.918,E2 -3242.918} C_VEL
LIN {X 0,Y 552.188,Z 185.7,A -85,B 0,C 180,E1 -3245.844,E2 -3245.844} C_VEL
LIN {X 0,Y 552.137,Z 185.704,A -85,B 0,C 180,E1 -3248.786,E2 -3248.786} C_VEL
LIN {X 0,Y 552.16,Z 185.704,A -85,B 0,C 180,E1 -3251.751,E2 -3251.751} C_VEL
LIN {X 0,Y 552.132,Z 185.704,A -85,B 0,C 180,E1 -3254.749,E2 -3254.749} C_VEL
LIN {X 0,Y 552.082,Z 185.717,A -85,B 0,C 180,E1 -3257.79,E2 -3257.79} C_VEL
LIN {X 0,Y 552.122,Z 185.711,A -85,B 0,C 180,E1 -3260.102,E2 -3260.102} C_VEL
LIN {X 0,Y 552.086,Z 185.711,A -85,B 0,C 180,E1 -3262.451,E2 -3262.451} C_VEL
LIN {X 0,Y 552.086,Z 185.713,A -85,B 0,C 180,E1 -3265.334,E2 -3265.334} C_VEL
LIN {X 0,Y 552.06,Z 185.716,A -85,B 0,C 180,E1 -3268.101,E2 -3268.101} C_VEL
LIN {X 0,Y 552.094,Z 185.708,A -85,B 0,C 180,E1 -3270.61,E2 -3270.61} C_VEL
LIN {X 0,Y 552.107,Z 185.71,A -85,B 0,C 180,E1 -3273.187,E2 -3273.187} C_VEL
LIN {X 0,Y 552.073,Z 185.715,A -85,B 0,C 180,E1 -3275.845,E2 -3275.845} C_VEL
LIN {X 0,Y 552.115,Z 185.706,A -85,B 0,C 180,E1 -3278.589,E2 -3278.589} C_VEL
LIN {X 0,Y 552.077,Z 185.719,A -85,B 0,C 180,E1 -3281.45,E2 -3281.45} C_VEL
LIN {X 0,Y 552.077,Z 185.711,A -85,B 0,C 180,E1 -3284.529,E2 -3284.529} C_VEL
LIN {X 0,Y 552.088,Z 185.713,A -85,B 0,C 180,E1 -3287.59,E2 -3287.59} C_VEL
LIN {X 0,Y 552.127,Z 185.705,A -85,B 0,C 180,E1 -3290.472,E2 -3290.472} C_VEL
LIN {X 0,Y 552.101,Z 185.714,A -85,B 0,C 180,E1 -3293.318,E2 -3293.318} C_VEL
LIN {X 0,Y 552.1,Z 185.708,A -85,B 0,C 180,E1 -3295.937,E2 -3295.937} C_VEL
LIN {X 0,Y 552.106,Z 185.711,A -85,B 0,C 180,E1 -3298.539,E2 -3298.539} C_VEL
LIN {X 0,Y 552.081,Z 185.714,A -85,B 0,C 180,E1 -3301.447,E2 -3301.447} C_VEL
LIN {X 0,Y 552.135,Z 185.726,A -85,B 0,C 180,E1 -3304.522,E2 -3304.522} C_VEL
LIN {X 0,Y 553.434,Z 193.407,A -85,B 0,C 180,E1 -3305.624,E2 -3305.624} C_VEL
LIN {X 0,Y 553.12,Z 212.388,A -85,B 0,C 180,E1 -3308.163,E2 -3308.163} C_VEL
LIN {X 0,Y 552.867,Z 233.165,A -85,B 0,C 180,E1 -3310.893,E2 -3310.893} C_VEL
LIN {X 0,Y 552.601,Z 255.181,A -85,B 0,C 180,E1 -3313.752,E2 -3313.752} C_VEL
LIN {X 0,Y 552.431,Z 269.72,A -85,B 0,C 180,E1 -3315.624,E2 -3315.624} C_VEL
LIN {X 0,Y 553.41,Z 277.829,A -85,B 0,C 180,E1 -3315.756,E2 -3315.756} C_VEL
LIN {X 0,Y 553.127,Z 378.767,A -85,B 0,C 180,E1 -3317.082,E2 -3317.082} C_VEL
LIN {X 0,Y 552.98,Z 392.121,A -85,B 0,C 180,E1 -3317.406,E2 -3317.406} C_VEL
LIN {X 0,Y 552.829,Z 404.35,A -85,B 0,C 180,E1 -3317.845,E2 -3317.845} C_VEL
LIN {X 0,Y 552.63,Z 416.298,A -85,B 0,C 180,E1 -3318.427,E2 -3318.427} C_VEL
LIN {X 0,Y 552.476,Z 428.189,A -85,B 0,C 180,E1 -3319.185,E2 -3319.185} C_VEL
LIN {X 0,Y 552.303,Z 438.602,A -85,B 0,C 180,E1 -3320.016,E2 -3320.016} C_VEL
LIN {X 0,Y 552.131,Z 447.111,A -85,B 0,C 180,E1 -3320.845,E2 -3320.845} C_VEL
LIN {X 0,Y 552.013,Z 454.959,A -85,B 0,C 180,E1 -3321.765,E2 -3321.765} C_VEL
LIN {X 0,Y 551.89,Z 462.62,A -85,B 0,C 180,E1 -3322.867,E2 -3322.867} C_VEL
LIN {X 0,Y 551.867,Z 469.678,A -85,B 0,C 180,E1 -3324.152,E2 -3324.152} C_VEL
LIN {X 0,Y 551.725,Z 474.372,A -85,B 0,C 180,E1 -3325.25,E2 -3325.25} C_VEL
LIN {X 0,Y 551.75,Z 477.957,A -85,B 0,C 180,E1 -3326.348,E2 -3326.348} C_VEL
LIN {X 0,Y 551.723,Z 479.806,A -85,B 0,C 180,E1 -3327.079,E2 -3327.079} C_VEL
LIN {X 0,Y 551.645,Z 482.182,A -85,B 0,C 180,E1 -3328.54,E2 -3328.54} C_VEL
LIN {X 0,Y 551.64,Z 483,A -85,B 0,C 180,E1 -3330,E2 -3330} C_VEL
LIN {X 0,Y 551.645,Z 482.184,A -85,B 0,C 180,E1 -3331.46,E2 -3331.46} C_VEL
LIN {X 0,Y 551.723,Z 479.81,A -85,B 0,C 180,E1 -3332.92,E2 -3332.92} C_VEL
LIN {X 0,Y 551.764,Z 476.896,A -85,B 0,C 180,E1 -3334.017,E2 -3334.017} C_VEL
LIN {X 0,Y 551.723,Z 472.949,A -85,B 0,C 180,E1 -3335.116,E2 -3335.116} C_VEL
LIN {X 0,Y 551.801,Z 467.198,A -85,B 0,C 180,E1 -3336.34,E2 -3336.34} C_VEL
LIN {X 0,Y 551.926,Z 460.237,A -85,B 0,C 180,E1 -3337.499,E2 -3337.499} C_VEL
LIN {X 0,Y 552.082,Z 451.993,A -85,B 0,C 180,E1 -3338.602,E2 -3338.602} C_VEL
LIN {X 0,Y 552.2,Z 443.542,A -85,B 0,C 180,E1 -3339.523,E2 -3339.523} C_VEL
LIN {X 0,Y 552.428,Z 433.093,A -85,B 0,C 180,E1 -3340.445,E2 -3340.445} C_VEL
LIN {X 0,Y 552.595,Z 422.288,A -85,B 0,C 180,E1 -3341.213,E2 -3341.213} C_VEL
LIN {X 0,Y 552.751,Z 411.406,A -85,B 0,C 180,E1 -3341.831,E2 -3341.831} C_VEL
LIN {X 0,Y 552.904,Z 399.73,A -85,B 0,C 180,E1 -3342.339,E2 -3342.339} C_VEL
LIN {X 0,Y 553.053,Z 386.213,A -85,B 0,C 180,E1 -3342.756,E2 -3342.756} C_VEL
LIN {X 0,Y 553.163,Z 372.847,A -85,B 0,C 180,E1 -3343.01,E2 -3343.01} C_VEL
LIN {X 0,Y 553.314,Z 275.919,A -85,B 0,C 180,E1 -3344.27,E2 -3344.27} C_VEL
LIN {X 0,Y 552.415,Z 269.489,A -85,B 0,C 180,E1 -3344.388,E2 -3344.388} C_VEL
LIN {X 0,Y 552.634,Z 247.076,A -85,B 0,C 180,E1 -3347.249,E2 -3347.249} C_VEL
LIN {X 0,Y 552.887,Z 225.149,A -85,B 0,C 180,E1 -3350.072,E2 -3350.072} C_VEL
LIN {X 0,Y 553.112,Z 202.678,A -85,B 0,C 180,E1 -3352.999,E2 -3352.999} C_VEL
LIN {X 0,Y 553.157,Z 191.997,A -85,B 0,C 180,E1 -3354.388,E2 -3354.388} C_VEL
LIN {X 0,Y 552.133,Z 185.713,A -85,B 0,C 180,E1 -3355.262,E2 -3355.262} C_VEL
LIN {X 0,Y 552.057,Z 185.716,A -85,B 0,C 180,E1 -3358.101,E2 -3358.101} C_VEL
LIN {X 0,Y 552.089,Z 185.715,A -85,B 0,C 180,E1 -3360.61,E2 -3360.61} C_VEL
LIN {X 0,Y 552.104,Z 185.714,A -85,B 0,C 180,E1 -3363.186,E2 -3363.186} C_VEL
LIN {X 0,Y 552.075,Z 185.711,A -85,B 0,C 180,E1 -3365.844,E2 -3365.844} C_VEL
LIN {X 0,Y 552.113,Z 185.713,A -85,B 0,C 180,E1 -3368.589,E2 -3368.589} C_VEL
LIN {X 0,Y 552.11,Z 185.707,A -85,B 0,C 180,E1 -3371.447,E2 -3371.447} C_VEL
LIN {X 0,Y 552.076,Z 185.719,A -85,B 0,C 180,E1 -3374.529,E2 -3374.529} C_VEL
LIN {X 0,Y 552.108,Z 185.706,A -85,B 0,C 180,E1 -3377.587,E2 -3377.587} C_VEL
LIN {X 0,Y 552.127,Z 185.713,A -85,B 0,C 180,E1 -3380.472,E2 -3380.472} C_VEL
LIN {X 0,Y 552.099,Z 185.708,A -85,B 0,C 180,E1 -3383.318,E2 -3383.318} C_VEL
LIN {X 0,Y 552.125,Z 185.708,A -85,B 0,C 180,E1 -3385.939,E2 -3385.939} C_VEL
LIN {X 0,Y 552.12,Z 185.71,A -85,B 0,C 180,E1 -3388.54,E2 -3388.54} C_VEL
LIN {X 0,Y 552.102,Z 185.708,A -85,B 0,C 180,E1 -3391.442,E2 -3391.442} C_VEL
LIN {X 0,Y 552.104,Z 185.709,A -85,B 0,C 180,E1 -3393.543,E2 -3393.543} C_VEL
LIN {X 0,Y 552.092,Z 185.709,A -85,B 0,C 180,E1 -3396.757,E2 -3396.757} C_VEL
LIN {X 0,Y 552.117,Z 185.706,A -85,B 0,C 180,E1 -3399.12,E2 -3399.12} C_VEL
LIN {X 0,Y 552.087,Z 185.713,A -85,B 0,C 180,E1 -3401.443,E2 -3401.443} C_VEL
LIN {X 0,Y 552.095,Z 185.716,A -85,B 0,C 180,E1 -3403.737,E2 -3403.737} C_VEL
LIN {X 0,Y 552.129,Z 185.71,A -85,B 0,C 180,E1 -3406.004,E2 -3406.004} C_VEL
LIN {X 0,Y 552.163,Z 185.701,A -85,B 0,C 180,E1 -3408.993,E2 -3408.993} C_VEL
LIN {X 0,Y 552.154,Z 185.705,A -85,B 0,C 180,E1 -3411.951,E2 -3411.951} C_VEL
LIN {X 0,Y 552.228,Z 185.694,A -85,B 0,C 180,E1 -3414.889,E2 -3414.889} C_VEL
LIN {X 0,Y 552.228,Z 185.695,A -85,B 0,C 180,E1 -3417.812,E2 -3417.812} C_VEL
LIN {X 0,Y 552.237,Z 185.693,A -85,B 0,C 180,E1 -3420.729,E2 -3420.729} C_VEL
LIN {X 0,Y 552.2,Z 185.7,A -85,B 0,C 180,E1 -3422.918,E2 -3422.918} C_VEL
LIN {X 0,Y 552.201,Z 185.697,A -85,B 0,C 180,E1 -3425.844,E2 -3425.844} C_VEL
LIN {X 0,Y 552.142,Z 185.708,A -85,B 0,C 180,E1 -3428.786,E2 -3428.786} C_VEL
LIN {X 0,Y 552.163,Z 185.703,A -85,B 0,C 180,E1 -3431.75,E2 -3431.75} C_VEL
LIN {X 0,Y 552.137,Z 185.712,A -85,B 0,C 180,E1 -3434.748,E2 -3434.748} C_VEL
LIN {X 0,Y 552.098,Z 185.71,A -85,B 0,C 180,E1 -3437.789,E2 -3437.789} C_VEL
LIN {X 0,Y 552.127,Z 185.707,A -85,B 0,C 180,E1 -3440.101,E2 -3440.101} C_VEL
LIN {X 0,Y 552.126,Z 185.849,A -85,B 0,C 180,E1 -3442.154,E2 -3442.154} C_VEL
LIN {X 0,Y 552.171,Z 191.468,A -85,B 0,C 180,E1 -3443.239,E2 -3443.239} C_VEL
LIN {X 0,Y 552.152,Z 193.876,A -85,B 0,C 180,E1 -3443.702,E2 -3443.702} C_VEL
LIN {X 0,Y 553.418,Z 201.773,A -85,B 0,C 180,E1 -3443.84,E2 -3443.84} C_VEL
LIN {X 0,Y 553.192,Z 285.344,A -85,B 0,C 180,E1 -3444.932,E2 -3444.932} C_VEL
LIN {X 0,Y 552.505,Z 291.193,A -85,B 0,C 180,E1 -3444.992,E2 -3444.992} C_VEL
LIN {X 0,Y 549.596,Z 300.671,A -85,B 0,C 180,E1 -3445.072,E2 -3445.072} C_VEL
LIN {X 0,Y 546.732,Z 310.029,A -85,B 0,C 180,E1 -3445.219,E2 -3445.219} C_VEL
LIN {X 0,Y 546.062,Z 315.678,A -85,B 0,C 180,E1 -3445.377,E2 -3445.377} C_VEL
LIN {X 0,Y 545.879,Z 328.175,A -85,B 0,C 180,E1 -3445.871,E2 -3445.871} C_VEL
LIN {X 0,Y 545.654,Z 339.806,A -85,B 0,C 180,E1 -3446.485,E2 -3446.485} C_VEL
LIN {X 0,Y 545.448,Z 351.065,A -85,B 0,C 180,E1 -3447.246,E2 -3447.246} C_VEL
LIN {X 0,Y 545.277,Z 360.732,A -85,B 0,C 180,E1 -3448.063,E2 -3448.063} C_VEL
LIN {X 0,Y 545.139,Z 369.829,A -85,B 0,C 180,E1 -3449.008,E2 -3449.008} C_VEL
LIN {X 0,Y 544.963,Z 377.552,A -85,B 0,C 180,E1 -3449.982,E2 -3449.982} C_VEL
LIN {X 0,Y 544.836,Z 384.547,A -85,B 0,C 180,E1 -3451.062,E2 -3451.062} C_VEL
LIN {X 0,Y 544.761,Z 390.232,A -85,B 0,C 180,E1 -3452.152,E2 -3452.152} C_VEL
LIN {X 0,Y 544.662,Z 395.038,A -85,B 0,C 180,E1 -3453.318,E2 -3453.318} C_VEL
LIN {X 0,Y 544.609,Z 398.926,A -85,B 0,C 180,E1 -3454.597,E2 -3454.597} C_VEL
LIN {X 0,Y 544.564,Z 401.086,A -85,B 0,C 180,E1 -3455.604,E2 -3455.604} C_VEL
LIN {X 0,Y 544.562,Z 402.716,A -85,B 0,C 180,E1 -3456.855,E2 -3456.855} C_VEL
LIN {X 0,Y 544.526,Z 403.177,A -85,B 0,C 180,E1 -3458.281,E2 -3458.281} C_VEL
LIN {X 0,Y 544.543,Z 402.698,A -85,B 0,C 180,E1 -3459.252,E2 -3459.252} C_VEL
LIN {X 0,Y 544.569,Z 401.212,A -85,B 0,C 180,E1 -3460.41,E2 -3460.41} C_VEL
LIN {X 0,Y 544.643,Z 398.78,A -85,B 0,C 180,E1 -3461.546,E2 -3461.546} C_VEL
LIN {X 0,Y 544.668,Z 395.438,A -85,B 0,C 180,E1 -3462.652,E2 -3462.652} C_VEL
LIN {X 0,Y 544.724,Z 390.297,A -85,B 0,C 180,E1 -3463.92,E2 -3463.92} C_VEL
LIN {X 0,Y 544.826,Z 383.539,A -85,B 0,C 180,E1 -3465.192,E2 -3465.192} C_VEL
LIN {X 0,Y 544.973,Z 376.596,A -85,B 0,C 180,E1 -3466.235,E2 -3466.235} C_VEL
LIN {X 0,Y 545.147,Z 367.916,A -85,B 0,C 180,E1 -3467.294,E2 -3467.294} C_VEL
LIN {X 0,Y 545.294,Z 359.054,A -85,B 0,C 180,E1 -3468.174,E2 -3468.174} C_VEL
LIN {X 0,Y 545.485,Z 347.868,A -85,B 0,C 180,E1 -3469.072,E2 -3469.072} C_VEL
LIN {X 0,Y 545.728,Z 336.26,A -85,B 0,C 180,E1 -3469.806,E2 -3469.806} C_VEL
LIN {X 0,Y 545.959,Z 323.488,A -85,B 0,C 180,E1 -3470.419,E2 -3470.419} C_VEL
LIN {X 0,Y 546.119,Z 310.534,A -85,B 0,C 180,E1 -3470.869,E2 -3470.869} C_VEL
LIN {X 0,Y 546.221,Z 297.61,A -85,B 0,C 180,E1 -3471.155,E2 -3471.155} C_VEL
LIN {X 0,Y 546.499,Z 201.563,A -85,B 0,C 180,E1 -3472.436,E2 -3472.436} C_VEL
LIN {X 0,Y 545.152,Z 194.143,A -85,B 0,C 180,E1 -3472.589,E2 -3472.589} C_VEL
LIN {X 0,Y 545.113,Z 186.583,A -85,B 0,C 180,E1 -3474.149,E2 -3474.149} C_VEL
LIN {X 0,Y 545.064,Z 186.594,A -85,B 0,C 180,E1 -3477.211,E2 -3477.211} C_VEL
LIN {X 0,Y 545.062,Z 186.586,A -85,B 0,C 180,E1 -3479.811,E2 -3479.811} C_VEL
LIN {X 0,Y 545.059,Z 186.585,A -85,B 0,C 180,E1 -3482.343,E2 -3482.343} C_VEL
LIN {X 0,Y 545.063,Z 186.589,A -85,B 0,C 180,E1 -3484.818,E2 -3484.818} C_VEL
LIN {X 0,Y 545.032,Z 186.594,A -85,B 0,C 180,E1 -3487.242,E2 -3487.242} C_VEL
LIN {X 0,Y 545.117,Z 186.579,A -85,B 0,C 180,E1 -3490.415,E2 -3490.415} C_VEL
LIN {X 0,Y 545.056,Z 186.587,A -85,B 0,C 180,E1 -3493.521,E2 -3493.521} C_VEL
LIN {X 0,Y 545.085,Z 186.581,A -85,B 0,C 180,E1 -3495.82,E2 -3495.82} C_VEL
LIN {X 0,Y 545.118,Z 186.586,A -85,B 0,C 180,E1 -3498.85,E2 -3498.85} C_VEL
LIN {X 0,Y 545.098,Z 186.58,A -85,B 0,C 180,E1 -3501.847,E2 -3501.847} C_VEL
LIN {X 0,Y 545.199,Z 186.574,A -85,B 0,C 180,E1 -3504.823,E2 -3504.823} C_VEL
LIN {X 0,Y 545.196,Z 186.568,A -85,B 0,C 180,E1 -3507.784,E2 -3507.784} C_VEL
LIN {X 0,Y 545.211,Z 186.571,A -85,B 0,C 180,E1 -3510.739,E2 -3510.739} C_VEL
LIN {X 0,Y 545.158,Z 186.575,A -85,B 0,C 180,E1 -3512.956,E2 -3512.956} C_VEL
LIN {X 0,Y 545.165,Z 186.575,A -85,B 0,C 180,E1 -3515.92,E2 -3515.92} C_VEL
LIN {X 0,Y 545.108,Z 186.58,A -85,B 0,C 180,E1 -3518.9,E2 -3518.9} C_VEL
LIN {X 0,Y 545.106,Z 186.583,A -85,B 0,C 180,E1 -3521.905,E2 -3521.905} C_VEL
LIN {X 0,Y 545.083,Z 186.582,A -85,B 0,C 180,E1 -3524.944,E2 -3524.944} C_VEL
LIN {X 0,Y 545.058,Z 186.594,A -85,B 0,C 180,E1 -3528.027,E2 -3528.027} C_VEL
LIN {X 0,Y 545.093,Z 186.585,A -85,B 0,C 180,E1 -3530.372,E2 -3530.372} C_VEL
LIN {X 0,Y 545.076,Z 186.586,A -85,B 0,C 180,E1 -3533.56,E2 -3533.56} C_VEL
LIN {X 0,Y 545.061,Z 186.584,A -85,B 0,C 180,E1 -3536.827,E2 -3536.827} C_VEL
LIN {X 0,Y 545.044,Z 186.589,A -85,B 0,C 180,E1 -3539.34,E2 -3539.34} C_VEL
LIN {X 0,Y 545.056,Z 186.592,A -85,B 0,C 180,E1 -3541.915,E2 -3541.915} C_VEL
LIN {X 0,Y 545.063,Z 186.584,A -85,B 0,C 180,E1 -3544.565,E2 -3544.565} C_VEL
LIN {X 0,Y 545.032,Z 186.593,A -85,B 0,C 180,E1 -3547.305,E2 -3547.305} C_VEL
LIN {X 0,Y 545.066,Z 186.585,A -85,B 0,C 180,E1 -3550.143,E2 -3550.143} C_VEL
LIN {X 0,Y 545.047,Z 186.59,A -85,B 0,C 180,E1 -3553.11,E2 -3553.11} C_VEL
LIN {X 0,Y 545.048,Z 186.586,A -85,B 0,C 180,E1 -3556.227,E2 -3556.227} C_VEL
LIN {X 0,Y 545.073,Z 186.586,A -85,B 0,C 180,E1 -3558.885,E2 -3558.885} C_VEL
LIN {X 0,Y 545.047,Z 186.588,A -85,B 0,C 180,E1 -3561.865,E2 -3561.865} C_VEL
LIN {X 0,Y 545.032,Z 186.589,A -85,B 0,C 180,E1 -3564.531,E2 -3564.531} C_VEL
LIN {X 0,Y 545.064,Z 186.593,A -85,B 0,C 180,E1 -3567.211,E2 -3567.211} C_VEL
LIN {X 0,Y 545.064,Z 186.585,A -85,B 0,C 180,E1 -3569.81,E2 -3569.81} C_VEL
LIN {X 0,Y 545.06,Z 186.591,A -85,B 0,C 180,E1 -3572.834,E2 -3572.834} C_VEL
LIN {X 0,Y 545.023,Z 186.59,A -85,B 0,C 180,E1 -3575.629,E2 -3575.629} C_VEL
LIN {X 0,Y 545.068,Z 186.585,A -85,B 0,C 180,E1 -3578.181,E2 -3578.181} C_VEL
LIN {X 0,Y 545.119,Z 186.581,A -85,B 0,C 180,E1 -3580.415,E2 -3580.415} C_VEL
LIN {X 0,Y 545.047,Z 186.587,A -85,B 0,C 180,E1 -3583.52,E2 -3583.52} C_VEL
LIN {X 0,Y 545.074,Z 186.583,A -85,B 0,C 180,E1 -3585.819,E2 -3585.819} C_VEL
LIN {X 0,Y 545.119,Z 186.583,A -85,B 0,C 180,E1 -3588.849,E2 -3588.849} C_VEL
LIN {X 0,Y 545.096,Z 186.581,A -85,B 0,C 180,E1 -3591.847,E2 -3591.847} C_VEL
LIN {X 0,Y 545.191,Z 186.573,A -85,B 0,C 180,E1 -3594.823,E2 -3594.823} C_VEL
LIN {X 0,Y 545.195,Z 186.569,A -85,B 0,C 180,E1 -3597.784,E2 -3597.784} C_VEL
LIN {X 0,Y 545.207,Z 186.57,A -85,B 0,C 180,E1 -3600.739,E2 -3600.739} C_VEL
LIN {X 0,Y 545.153,Z 186.574,A -85,B 0,C 180,E1 -3602.956,E2 -3602.956} C_VEL
LIN {X 0,Y 545.137,Z 186.58,A -85,B 0,C 180,E1 -3605.92,E2 -3605.92} C_VEL
LIN {X 0,Y 545.098,Z 186.581,A -85,B 0,C 180,E1 -3608.9,E2 -3608.9} C_VEL
LIN {X 0,Y 545.103,Z 186.586,A -85,B 0,C 180,E1 -3611.905,E2 -3611.905} C_VEL
LIN {X 0,Y 545.083,Z 186.582,A -85,B 0,C 180,E1 -3614.944,E2 -3614.944} C_VEL
LIN {X 0,Y 545.052,Z 186.594,A -85,B 0,C 180,E1 -3618.027,E2 -3618.027} C_VEL
LIN {X 0,Y 545.087,Z 186.584,A -85,B 0,C 180,E1 -3620.373,E2 -3620.373} C_VEL
LIN {X 0,Y 545.074,Z 186.589,A -85,B 0,C 180,E1 -3623.56,E2 -3623.56} C_VEL
LIN {X 0,Y 545.058,Z 186.585,A -85,B 0,C 180,E1 -3626.827,E2 -3626.827} C_VEL
LIN {X 0,Y 545.029,Z 186.593,A -85,B 0,C 180,E1 -3629.341,E2 -3629.341} C_VEL
LIN {X 0,Y 545.055,Z 186.59,A -85,B 0,C 180,E1 -3631.915,E2 -3631.915} C_VEL
LIN {X 0,Y 545.049,Z 186.586,A -85,B 0,C 180,E1 -3634.566,E2 -3634.566} C_VEL
LIN {X 0,Y 545.032,Z 186.595,A -85,B 0,C 180,E1 -3637.305,E2 -3637.305} C_VEL
LIN {X 0,Y 545.065,Z 186.585,A -85,B 0,C 180,E1 -3640.143,E2 -3640.143} C_VEL
LIN {X 0,Y 545.02,Z 186.595,A -85,B 0,C 180,E1 -3643.113,E2 -3643.113} C_VEL
LIN {X 0,Y 545.03,Z 186.588,A -85,B 0,C 180,E1 -3646.229,E2 -3646.229} C_VEL
LIN {X 0,Y 545.03,Z 186.593,A -85,B 0,C 180,E1 -3648.88,E2 -3648.88} C_VEL
LIN {X 0,Y 545.049,Z 186.587,A -85,B 0,C 180,E1 -3651.762,E2 -3651.762} C_VEL
LIN {X 0,Y 545.027,Z 186.591,A -85,B 0,C 180,E1 -3654.531,E2 -3654.531} C_VEL
LIN {X 0,Y 545.064,Z 186.591,A -85,B 0,C 180,E1 -3657.211,E2 -3657.211} C_VEL
LIN {X 0,Y 545.065,Z 186.585,A -85,B 0,C 180,E1 -3659.81,E2 -3659.81} C_VEL
LIN {X 0,Y 545.039,Z 186.596,A -85,B 0,C 180,E1 -3662.839,E2 -3662.839} C_VEL
LIN {X 0,Y 545.093,Z 186.639,A -85,B 0,C 180,E1 -3664.355,E2 -3664.355} C_VEL
LIN {X 0,Y 546.494,Z 194.466,A -85,B 0,C 180,E1 -3665.497,E2 -3665.497} C_VEL
LIN {X 0,Y 546.158,Z 213.56,A -85,B 0,C 180,E1 -3668.088,E2 -3668.088} C_VEL
LIN {X 0,Y 545.862,Z 234.188,A -85,B 0,C 180,E1 -3670.833,E2 -3670.833} C_VEL
LIN {X 0,Y 545.573,Z 256.204,A -85,B 0,C 180,E1 -3673.729,E2 -3673.729} C_VEL
LIN {X 0,Y 545.397,Z 269.252,A -85,B 0,C 180,E1 -3675.435,E2 -3675.435} C_VEL
LIN {X 0,Y 546.518,Z 278.887,A -85,B 0,C 180,E1 -3675.596,E2 -3675.596} C_VEL
LIN {X 0,Y 546.19,Z 377.974,A -85,B 0,C 180,E1 -3676.915,E2 -3676.915} C_VEL
LIN {X 0,Y 546.039,Z 391.434,A -85,B 0,C 180,E1 -3677.243,E2 -3677.243} C_VEL
LIN {X 0,Y 545.83,Z 404.845,A -85,B 0,C 180,E1 -3677.734,E2 -3677.734} C_VEL
LIN {X 0,Y 545.61,Z 416.657,A -85,B 0,C 180,E1 -3678.327,E2 -3678.327} C_VEL
LIN {X 0,Y 545.455,Z 427.794,A -85,B 0,C 180,E1 -3679.044,E2 -3679.044} C_VEL
LIN {X 0,Y 545.262,Z 438.323,A -85,B 0,C 180,E1 -3679.885,E2 -3679.885} C_VEL
LIN {X 0,Y 545.088,Z 446.934,A -85,B 0,C 180,E1 -3680.725,E2 -3680.725} C_VEL
LIN {X 0,Y 544.961,Z 454.884,A -85,B 0,C 180,E1 -3681.658,E2 -3681.658} C_VEL
LIN {X 0,Y 544.824,Z 462.615,A -85,B 0,C 180,E1 -3682.775,E2 -3682.775} C_VEL
LIN {X 0,Y 544.777,Z 469.678,A -85,B 0,C 180,E1 -3684.076,E2 -3684.076} C_VEL
LIN {X 0,Y 544.629,Z 474.372,A -85,B 0,C 180,E1 -3685.188,E2 -3685.188} C_VEL
LIN {X 0,Y 544.669,Z 477.957,A -85,B 0,C 180,E1 -3686.301,E2 -3686.301} C_VEL
LIN {X 0,Y 544.65,Z 479.806,A -85,B 0,C 180,E1 -3687.041,E2 -3687.041} C_VEL
LIN {X 0,Y 544.546,Z 482.181,A -85,B 0,C 180,E1 -3688.521,E2 -3688.521} C_VEL
LIN {X 0,Y 544.541,Z 483,A -85,B 0,C 180,E1 -3690,E2 -3690} C_VEL
LIN {X 0,Y 544.546,Z 482.183,A -85,B 0,C 180,E1 -3691.479,E2 -3691.479} C_VEL
LIN {X 0,Y 544.65,Z 479.81,A -85,B 0,C 180,E1 -3692.958,E2 -3692.958} C_VEL
LIN {X 0,Y 544.684,Z 476.896,A -85,B 0,C 180,E1 -3694.069,E2 -3694.069} C_VEL
LIN {X 0,Y 544.653,Z 472.949,A -85,B 0,C 180,E1 -3695.182,E2 -3695.182} C_VEL
LIN {X 0,Y 544.738,Z 467.713,A -85,B 0,C 180,E1 -3696.326,E2 -3696.326} C_VEL
LIN {X 0,Y 544.836,Z 461.458,A -85,B 0,C 180,E1 -3697.411,E2 -3697.411} C_VEL
LIN {X 0,Y 545.006,Z 453.384,A -85,B 0,C 180,E1 -3698.528,E2 -3698.528} C_VEL
LIN {X 0,Y 545.113,Z 445.123,A -85,B 0,C 180,E1 -3699.461,E2 -3699.461} C_VEL
LIN {X 0,Y 545.357,Z 435.061,A -85,B 0,C 180,E1 -3700.394,E2 -3700.394} C_VEL
LIN {X 0,Y 545.565,Z 424.116,A -85,B 0,C 180,E1 -3701.208,E2 -3701.208} C_VEL
LIN {X 0,Y 545.714,Z 412.554,A -85,B 0,C 180,E1 -3701.891,E2 -3701.891} C_VEL
LIN {X 0,Y 545.918,Z 400.215,A -85,B 0,C 180,E1 -3702.453,E2 -3702.453} C_VEL
LIN {X 0,Y 546.079,Z 387.213,A -85,B 0,C 180,E1 -3702.874,E2 -3702.874} C_VEL
LIN {X 0,Y 546.218,Z 373.376,A -85,B 0,C 180,E1 -3703.154,E2 -3703.154} C_VEL
LIN {X 0,Y 546.426,Z 276.922,A -85,B 0,C 180,E1 -3704.428,E2 -3704.428} C_VEL
LIN {X 0,Y 545.341,Z 268.975,A -85,B 0,C 180,E1 -3704.567,E2 -3704.567} C_VEL
LIN {X 0,Y 545.605,Z 247.264,A -85,B 0,C 180,E1 -3707.365,E2 -3707.365} C_VEL
LIN {X 0,Y 545.873,Z 226.279,A -85,B 0,C 180,E1 -3710.102,E2 -3710.102} C_VEL
LIN {X 0,Y 546.152,Z 204.96,A -85,B 0,C 180,E1 -3712.909,E2 -3712.909} C_VEL
LIN {X 0,Y 546.143,Z 192.748,A -85,B 0,C 180,E1 -3714.52,E2 -3714.52} C_VEL
LIN {X 0,Y 545.079,Z 186.592,A -85,B 0,C 180,E1 -3715.384,E2 -3715.384} C_VEL
LIN {X 0,Y 545.04,Z 186.592,A -85,B 0,C 180,E1 -3718.496,E2 -3718.496} C_VEL
LIN {X 0,Y 545.053,Z 186.595,A -85,B 0,C 180,E1 -3721.049,E2 -3721.049} C_VEL
LIN {X 0,Y 545.048,Z 186.588,A -85,B 0,C 180,E1 -3723.673,E2 -3723.673} C_VEL
LIN {X 0,Y 545.065,Z 186.592,A -85,B 0,C 180,E1 -3726.925,E2 -3726.925} C_VEL
LIN {X 0,Y 545.063,Z 186.586,A -85,B 0,C 180,E1 -3730.143,E2 -3730.143} C_VEL
LIN {X 0,Y 545.039,Z 186.595,A -85,B 0,C 180,E1 -3732.694,E2 -3732.694} C_VEL
LIN {X 0,Y 545.03,Z 186.59,A -85,B 0,C 180,E1 -3735.17,E2 -3735.17} C_VEL
LIN {X 0,Y 545.061,Z 186.585,A -85,B 0,C 180,E1 -3737.895,E2 -3737.895} C_VEL
LIN {X 0,Y 545.077,Z 186.587,A -85,B 0,C 180,E1 -3740.818,E2 -3740.818} C_VEL
LIN {X 0,Y 545.034,Z 186.589,A -85,B 0,C 180,E1 -3743.619,E2 -3743.619} C_VEL
LIN {X 0,Y 545.064,Z 186.593,A -85,B 0,C 180,E1 -3746.328,E2 -3746.328} C_VEL
LIN {X 0,Y 545.064,Z 186.585,A -85,B 0,C 180,E1 -3748.952,E2 -3748.952} C_VEL
LIN {X 0,Y 545.081,Z 186.583,A -85,B 0,C 180,E1 -3751.506,E2 -3751.506} C_VEL
LIN {X 0,Y 545.062,Z 186.592,A -85,B 0,C 180,E1 -3753.998,E2 -3753.998} C_VEL
LIN {X 0,Y 545.034,Z 186.589,A -85,B 0,C 180,E1 -3757.242,E2 -3757.242} C_VEL
LIN {X 0,Y 545.116,Z 186.581,A -85,B 0,C 180,E1 -3760.415,E2 -3760.415} C_VEL
LIN {X 0,Y 545.047,Z 186.591,A -85,B 0,C 180,E1 -3763.52,E2 -3763.52} C_VEL
LIN {X 0,Y 545.083,Z 186.59,A -85,B 0,C 180,E1 -3765.82,E2 -3765.82} C_VEL
LIN {X 0,Y 545.119,Z 186.577,A -85,B 0,C 180,E1 -3768.849,E2 -3768.849} C_VEL
LIN {X 0,Y 545.125,Z 186.582,A -85,B 0,C 180,E1 -3771.847,E2 -3771.847} C_VEL
LIN {X 0,Y 545.204,Z 186.568,A -85,B 0,C 180,E1 -3774.823,E2 -3774.823} C_VEL
LIN {X 0,Y 545.199,Z 186.571,A -85,B 0,C 180,E1 -3777.784,E2 -3777.784} C_VEL
LIN {X 0,Y 545.208,Z 186.569,A -85,B 0,C 180,E1 -3780.739,E2 -3780.739} C_VEL
LIN {X 0,Y 545.168,Z 186.577,A -85,B 0,C 180,E1 -3782.956,E2 -3782.956} C_VEL
LIN {X 0,Y 545.171,Z 186.572,A -85,B 0,C 180,E1 -3785.919,E2 -3785.919} C_VEL
LIN {X 0,Y 545.102,Z 186.586,A -85,B 0,C 180,E1 -3788.9,E2 -3788.9} C_VEL
LIN {X 0,Y 545.136,Z 186.578,A -85,B 0,C 180,E1 -3791.904,E2 -3791.904} C_VEL
LIN {X 0,Y 545.086,Z 186.591,A -85,B 0,C 180,E1 -3794.944,E2 -3794.944} C_VEL
LIN {X 0,Y 545.07,Z 186.586,A -85,B 0,C 180,E1 -3798.026,E2 -3798.026} C_VEL
LIN {X 0,Y 545.093,Z 186.586,A -85,B 0,C 180,E1 -3800.372,E2 -3800.372} C_VEL
LIN {X 0,Y 545.111,Z 186.704,A -85,B 0,C 180,E1 -3802.08,E2 -3802.08} C_VEL
LIN {X 0,Y 545.157,Z 194.164,A -85,B 0,C 180,E1 -3803.505,E2 -3803.505} C_VEL
LIN {X 0,Y 546.568,Z 202.076,A -85,B 0,C 180,E1 -3803.658,E2 -3803.658} C_VEL
LIN {X 0,Y 546.221,Z 300.545,A -85,B 0,C 180,E1 -3804.985,E2 -3804.985} C_VEL
LIN {X 0,Y 546.06,Z 313.662,A -85,B 0,C 180,E1 -3805.314,E2 -3805.314} C_VEL
LIN {X 0,Y 546.062,Z 315.678,A -85,B 0,C 180,E1 -3805.377,E2 -3805.377} C_VEL
LIN {X 0,Y 545.328,Z 321.281,A -85,B 0,C 180,E1 -3805.56,E2 -3805.56} C_VEL
LIN {X 0,Y 542.406,Z 330.28,A -85,B 0,C 180,E1 -3805.879,E2 -3805.879} C_VEL
LIN {X 0,Y 539.41,Z 338.96,A -85,B 0,C 180,E1 -3806.271,E2 -3806.271} C_VEL
LIN {X 0,Y 538.668,Z 344.054,A -85,B 0,C 180,E1 -3806.576,E2 -3806.576} C_VEL
LIN {X 0,Y 538.398,Z 355.461,A -85,B 0,C 180,E1 -3807.422,E2 -3807.422} C_VEL
LIN {X 0,Y 538.225,Z 365.499,A -85,B 0,C 180,E1 -3808.358,E2 -3808.358} C_VEL
LIN {X 0,Y 538.007,Z 373.981,A -85,B 0,C 180,E1 -3809.331,E2 -3809.331} C_VEL
LIN {X 0,Y 537.89,Z 381.707,A -85,B 0,C 180,E1 -3810.419,E2 -3810.419} C_VEL
LIN {X 0,Y 537.763,Z 388.031,A -85,B 0,C 180,E1 -3811.517,E2 -3811.517} C_VEL
LIN {X 0,Y 537.647,Z 393.883,A -85,B 0,C 180,E1 -3812.808,E2 -3812.808} C_VEL
LIN {X 0,Y 537.555,Z 398.528,A -85,B 0,C 180,E1 -3814.207,E2 -3814.207} C_VEL
LIN {X 0,Y 537.517,Z 400.75,A -85,B 0,C 180,E1 -3815.12,E2 -3815.12} C_VEL
LIN {X 0,Y 537.476,Z 402.336,A -85,B 0,C 180,E1 -3816.045,E2 -3816.045} C_VEL
LIN {X 0,Y 537.465,Z 403.407,A -85,B 0,C 180,E1 -3817.094,E2 -3817.094} C_VEL
LIN {X 0,Y 537.461,Z 403.69,A -85,B 0,C 180,E1 -3818.319,E2 -3818.319} C_VEL
LIN {X 0,Y 537.494,Z 402.603,A -85,B 0,C 180,E1 -3819.844,E2 -3819.844} C_VEL
LIN {X 0,Y 537.555,Z 399.933,A -85,B 0,C 180,E1 -3821.318,E2 -3821.318} C_VEL
LIN {X 0,Y 537.629,Z 395.546,A -85,B 0,C 180,E1 -3822.825,E2 -3822.825} C_VEL
LIN {X 0,Y 537.676,Z 390.6,A -85,B 0,C 180,E1 -3824.036,E2 -3824.036} C_VEL
LIN {X 0,Y 537.802,Z 384.082,A -85,B 0,C 180,E1 -3825.274,E2 -3825.274} C_VEL
LIN {X 0,Y 537.954,Z 376.643,A -85,B 0,C 180,E1 -3826.4,E2 -3826.4} C_VEL
LIN {X 0,Y 538.148,Z 367.961,A -85,B 0,C 180,E1 -3827.458,E2 -3827.458} C_VEL
LIN {X 0,Y 538.364,Z 358.602,A -85,B 0,C 180,E1 -3828.384,E2 -3828.384} C_VEL
LIN {X 0,Y 538.541,Z 347.549,A -85,B 0,C 180,E1 -3829.27,E2 -3829.27} C_VEL
LIN {X 0,Y 538.796,Z 336.492,A -85,B 0,C 180,E1 -3829.967,E2 -3829.967} C_VEL
LIN {X 0,Y 539.042,Z 324.867,A -85,B 0,C 180,E1 -3830.536,E2 -3830.536} C_VEL
LIN {X 0,Y 539.177,Z 311.564,A -85,B 0,C 180,E1 -3831.014,E2 -3831.014} C_VEL
LIN {X 0,Y 539.32,Z 298.414,A -85,B 0,C 180,E1 -3831.315,E2 -3831.315} C_VEL
LIN {X 0,Y 539.707,Z 202.885,A -85,B 0,C 180,E1 -3832.608,E2 -3832.608} C_VEL
LIN {X 0,Y 538.172,Z 194.486,A -85,B 0,C 180,E1 -3832.783,E2 -3832.783} C_VEL
LIN {X 0,Y 538.06,Z 187.462,A -85,B 0,C 180,E1 -3834.238,E2 -3834.238} C_VEL
LIN {X 0,Y 538.031,Z 187.464,A -85,B 0,C 180,E1 -3836.728,E2 -3836.728} C_VEL
LIN {X 0,Y 538.014,Z 187.467,A -85,B 0,C 180,E1 -3839.559,E2 -3839.559} C_VEL
LIN {X 0,Y 538.028,Z 187.461,A -85,B 0,C 180,E1 -3841.95,E2 -3841.95} C_VEL
LIN {X 0,Y 538.021,Z 187.463,A -85,B 0,C 180,E1 -3844.465,E2 -3844.465} C_VEL
LIN {X 0,Y 538.01,Z 187.47,A -85,B 0,C 180,E1 -3846.928,E2 -3846.928} C_VEL
LIN {X 0,Y 538.081,Z 187.454,A -85,B 0,C 180,E1 -3850.148,E2 -3850.148} C_VEL
LIN {X 0,Y 538.003,Z 187.467,A -85,B 0,C 180,E1 -3853.299,E2 -3853.299} C_VEL
LIN {X 0,Y 538.057,Z 187.457,A -85,B 0,C 180,E1 -3855.631,E2 -3855.631} C_VEL
LIN {X 0,Y 538.078,Z 187.463,A -85,B 0,C 180,E1 -3858.702,E2 -3858.702} C_VEL
LIN {X 0,Y 538.062,Z 187.456,A -85,B 0,C 180,E1 -3861.739,E2 -3861.739} C_VEL
LIN {X 0,Y 538.157,Z 187.452,A -85,B 0,C 180,E1 -3864.755,E2 -3864.755} C_VEL
LIN {X 0,Y 538.168,Z 187.444,A -85,B 0,C 180,E1 -3867.755,E2 -3867.755} C_VEL
LIN {X 0,Y 538.181,Z 187.447,A -85,B 0,C 180,E1 -3870.748,E2 -3870.748} C_VEL
LIN {X 0,Y 538.125,Z 187.45,A -85,B 0,C 180,E1 -3872.995,E2 -3872.995} C_VEL
LIN {X 0,Y 538.116,Z 187.454,A -85,B 0,C 180,E1 -3875.998,E2 -3875.998} C_VEL
LIN {X 0,Y 538.059,Z 187.457,A -85,B 0,C 180,E1 -3879.018,E2 -3879.018} C_VEL
LIN {X 0,Y 538.066,Z 187.463,A -85,B 0,C 180,E1 -3882.063,E2 -3882.063} C_VEL
LIN {X 0,Y 538.042,Z 187.459,A -85,B 0,C 180,E1 -3885.144,E2 -3885.144} C_VEL
LIN {X 0,Y 538.012,Z 187.469,A -85,B 0,C 180,E1 -3888.271,E2 -3888.271} C_VEL
LIN {X 0,Y 538.038,Z 187.461,A -85,B 0,C 180,E1 -3890.652,E2 -3890.652} C_VEL
LIN {X 0,Y 538.009,Z 187.472,A -85,B 0,C 180,E1 -3893.878,E2 -3893.878} C_VEL
LIN {X 0,Y 538.018,Z 187.464,A -85,B 0,C 180,E1 -3896.368,E2 -3896.368} C_VEL
LIN {X 0,Y 538.032,Z 187.46,A -85,B 0,C 180,E1 -3898.933,E2 -3898.933} C_VEL
LIN {X 0,Y 538.012,Z 187.47,A -85,B 0,C 180,E1 -3901.887,E2 -3901.887} C_VEL
LIN {X 0,Y 538.012,Z 187.463,A -85,B 0,C 180,E1 -3904.617,E2 -3904.617} C_VEL
LIN {X 0,Y 538.001,Z 187.467,A -85,B 0,C 180,E1 -3907.169,E2 -3907.169} C_VEL
LIN {X 0,Y 538.012,Z 187.468,A -85,B 0,C 180,E1 -3909.798,E2 -3909.798} C_VEL
LIN {X 0,Y 538.001,Z 187.465,A -85,B 0,C 180,E1 -3912.788,E2 -3912.788} C_VEL
LIN {X 0,Y 538,Z 187.469,A -85,B 0,C 180,E1 -3915.137,E2 -3915.137} C_VEL
LIN {X 0,Y 538.021,Z 187.462,A -85,B 0,C 180,E1 -3918.226,E2 -3918.226} C_VEL
LIN {X 0,Y 538.012,Z 187.47,A -85,B 0,C 180,E1 -3921.169,E2 -3921.169} C_VEL
LIN {X 0,Y 537.992,Z 187.465,A -85,B 0,C 180,E1 -3924.09,E2 -3924.09} C_VEL
LIN {X 0,Y 538.034,Z 187.463,A -85,B 0,C 180,E1 -3926.728,E2 -3926.728} C_VEL
LIN {X 0,Y 538.008,Z 187.466,A -85,B 0,C 180,E1 -3929.56,E2 -3929.56} C_VEL
LIN {X 0,Y 537.998,Z 187.464,A -85,B 0,C 180,E1 -3931.948,E2 -3931.948} C_VEL
LIN {X 0,Y 538.034,Z 187.462,A -85,B 0,C 180,E1 -3934.465,E2 -3934.465} C_VEL
LIN {X 0,Y 538.009,Z 187.472,A -85,B 0,C 180,E1 -3936.928,E2 -3936.928} C_VEL
LIN {X 0,Y 538.084,Z 187.455,A -85,B 0,C 180,E1 -3940.148,E2 -3940.148} C_VEL
LIN {X 0,Y 537.997,Z 187.467,A -85,B 0,C 180,E1 -3943.298,E2 -3943.298} C_VEL
LIN {X 0,Y 538.045,Z 187.458,A -85,B 0,C 180,E1 -3945.63,E2 -3945.63} C_VEL
LIN {X 0,Y 538.079,Z 187.463,A -85,B 0,C 180,E1 -3948.702,E2 -3948.702} C_VEL
LIN {X 0,Y 538.06,Z 187.457,A -85,B 0,C 180,E1 -3951.739,E2 -3951.739} C_VEL
LIN {X 0,Y 538.148,Z 187.451,A -85,B 0,C 180,E1 -3954.755,E2 -3954.755} C_VEL
LIN {X 0,Y 538.167,Z 187.444,A -85,B 0,C 180,E1 -3957.755,E2 -3957.755} C_VEL
LIN {X 0,Y 538.178,Z 187.445,A -85,B 0,C 180,E1 -3960.748,E2 -3960.748} C_VEL
LIN {X 0,Y 538.12,Z 187.45,A -85,B 0,C 180,E1 -3962.995,E2 -3962.995} C_VEL
LIN {X 0,Y 538.09,Z 187.459,A -85,B 0,C 180,E1 -3965.998,E2 -3965.998} C_VEL
LIN {X 0,Y 538.05,Z 187.458,A -85,B 0,C 180,E1 -3969.018,E2 -3969.018} C_VEL
LIN {X 0,Y 538.062,Z 187.466,A -85,B 0,C 180,E1 -3972.063,E2 -3972.063} C_VEL
LIN {X 0,Y 538.042,Z 187.459,A -85,B 0,C 180,E1 -3975.144,E2 -3975.144} C_VEL
LIN {X 0,Y 538.006,Z 187.468,A -85,B 0,C 180,E1 -3978.271,E2 -3978.271} C_VEL
LIN {X 0,Y 538.031,Z 187.461,A -85,B 0,C 180,E1 -3980.652,E2 -3980.652} C_VEL
LIN {X 0,Y 538.009,Z 187.464,A -85,B 0,C 180,E1 -3983.072,E2 -3983.072} C_VEL
LIN {X 0,Y 537.998,Z 187.472,A -85,B 0,C 180,E1 -3985.661,E2 -3985.661} C_VEL
LIN {X 0,Y 537.995,Z 187.469,A -85,B 0,C 180,E1 -3988.053,E2 -3988.053} C_VEL
LIN {X 0,Y 538.01,Z 187.463,A -85,B 0,C 180,E1 -3990.628,E2 -3990.628} C_VEL
LIN {X 0,Y 538.023,Z 187.466,A -85,B 0,C 180,E1 -3993.278,E2 -3993.278} C_VEL
LIN {X 0,Y 537.991,Z 187.468,A -85,B 0,C 180,E1 -3996.005,E2 -3996.005} C_VEL
LIN {X 0,Y 538.011,Z 187.464,A -85,B 0,C 180,E1 -3998.831,E2 -3998.831} C_VEL
LIN {X 0,Y 537.991,Z 187.468,A -85,B 0,C 180,E1 -4001.874,E2 -4001.874} C_VEL
LIN {X 0,Y 537.996,Z 187.468,A -85,B 0,C 180,E1 -4004.864,E2 -4004.864} C_VEL
LIN {X 0,Y 537.976,Z 187.476,A -85,B 0,C 180,E1 -4007.209,E2 -4007.209} C_VEL
LIN {X 0,Y 538.01,Z 187.463,A -85,B 0,C 180,E1 -4010.201,E2 -4010.201} C_VEL
LIN {X 0,Y 538.021,Z 187.471,A -85,B 0,C 180,E1 -4013.066,E2 -4013.066} C_VEL
LIN {X 0,Y 538,Z 187.464,A -85,B 0,C 180,E1 -4015.825,E2 -4015.825} C_VEL
LIN {X 0,Y 537.998,Z 187.468,A -85,B 0,C 180,E1 -4018.498,E2 -4018.498} C_VEL
LIN {X 0,Y 538.004,Z 187.472,A -85,B 0,C 180,E1 -4021.096,E2 -4021.096} C_VEL
LIN {X 0,Y 538.054,Z 187.572,A -85,B 0,C 180,E1 -4024.187,E2 -4024.187} C_VEL
LIN {X 0,Y 539.528,Z 195.518,A -85,B 0,C 180,E1 -4025.365,E2 -4025.365} C_VEL
LIN {X 0,Y 539.247,Z 213.109,A -85,B 0,C 180,E1 -4027.793,E2 -4027.793} C_VEL
LIN {X 0,Y 538.902,Z 233.743,A -85,B 0,C 180,E1 -4030.576,E2 -4030.576} C_VEL
LIN {X 0,Y 538.554,Z 254.296,A -85,B 0,C 180,E1 -4033.316,E2 -4033.316} C_VEL
LIN {X 0,Y 538.339,Z 268.781,A -85,B 0,C 180,E1 -4035.241,E2 -4035.241} C_VEL
LIN {X 0,Y 539.631,Z 279.658,A -85,B 0,C 180,E1 -4035.428,E2 -4035.428} C_VEL
LIN {X 0,Y 539.255,Z 378.364,A -85,B 0,C 180,E1 -4036.768,E2 -4036.768} C_VEL
LIN {X 0,Y 539.085,Z 391.511,A -85,B 0,C 180,E1 -4037.099,E2 -4037.099} C_VEL
LIN {X 0,Y 538.85,Z 404.201,A -85,B 0,C 180,E1 -4037.572,E2 -4037.572} C_VEL
LIN {X 0,Y 538.658,Z 414.964,A -85,B 0,C 180,E1 -4038.11,E2 -4038.11} C_VEL
LIN {X 0,Y 538.414,Z 427.208,A -85,B 0,C 180,E1 -4038.899,E2 -4038.899} C_VEL
LIN {X 0,Y 538.197,Z 437.751,A -85,B 0,C 180,E1 -4039.751,E2 -4039.751} C_VEL
LIN {X 0,Y 538.021,Z 446.375,A -85,B 0,C 180,E1 -4040.602,E2 -4040.602} C_VEL
LIN {X 0,Y 537.914,Z 454.338,A -85,B 0,C 180,E1 -4041.548,E2 -4041.548} C_VEL
LIN {X 0,Y 537.755,Z 462.113,A -85,B 0,C 180,E1 -4042.679,E2 -4042.679} C_VEL
LIN {X 0,Y 537.675,Z 469.28,A -85,B 0,C 180,E1 -4043.997,E2 -4043.997} C_VEL
LIN {X 0,Y 537.54,Z 474.043,A -85,B 0,C 180,E1 -4045.125,E2 -4045.125} C_VEL
LIN {X 0,Y 537.591,Z 477.694,A -85,B 0,C 180,E1 -4046.252,E2 -4046.252} C_VEL
LIN {X 0,Y 537.551,Z 479.572,A -85,B 0,C 180,E1 -4047.002,E2 -4047.002} C_VEL
LIN {X 0,Y 537.49,Z 480.978,A -85,B 0,C 180,E1 -4047.752,E2 -4047.752} C_VEL
LIN {X 0,Y 537.444,Z 482.595,A -85,B 0,C 180,E1 -4049.251,E2 -4049.251} C_VEL
LIN {X 0,Y 537.444,Z 482.813,A -85,B 0,C 180,E1 -4050,E2 -4050} C_VEL
LIN {X 0,Y 537.444,Z 482.594,A -85,B 0,C 180,E1 -4050.749,E2 -4050.749} C_VEL
LIN {X 0,Y 537.49,Z 480.978,A -85,B 0,C 180,E1 -4052.248,E2 -4052.248} C_VEL
LIN {X 0,Y 537.551,Z 479.571,A -85,B 0,C 180,E1 -4052.998,E2 -4052.998} C_VEL
LIN {X 0,Y 537.603,Z 476.606,A -85,B 0,C 180,E1 -4054.123,E2 -4054.123} C_VEL
LIN {X 0,Y 537.587,Z 472.585,A -85,B 0,C 180,E1 -4055.25,E2 -4055.25} C_VEL
LIN {X 0,Y 537.657,Z 466.411,A -85,B 0,C 180,E1 -4056.566,E2 -4056.566} C_VEL
LIN {X 0,Y 537.777,Z 459.654,A -85,B 0,C 180,E1 -4057.698,E2 -4057.698} C_VEL
LIN {X 0,Y 537.949,Z 451.278,A -85,B 0,C 180,E1 -4058.83,E2 -4058.83} C_VEL
LIN {X 0,Y 538.088,Z 442.684,A -85,B 0,C 180,E1 -4059.776,E2 -4059.776} C_VEL
LIN {X 0,Y 538.321,Z 432.077,A -85,B 0,C 180,E1 -4060.722,E2 -4060.722} C_VEL
LIN {X 0,Y 538.526,Z 420.775,A -85,B 0,C 180,E1 -4061.533,E2 -4061.533} C_VEL
LIN {X 0,Y 538.79,Z 410.075,A -85,B 0,C 180,E1 -4062.142,E2 -4062.142} C_VEL
LIN {X 0,Y 538.991,Z 398.211,A -85,B 0,C 180,E1 -4062.663,E2 -4062.663} C_VEL
LIN {X 0,Y 539.172,Z 385.459,A -85,B 0,C 180,E1 -4063.066,E2 -4063.066} C_VEL
LIN {X 0,Y 539.306,Z 372.388,A -85,B 0,C 180,E1 -4063.326,E2 -4063.326} C_VEL
LIN {X 0,Y 539.471,Z 276.804,A -85,B 0,C 180,E1 -4064.611,E2 -4064.611} C_VEL
LIN {X 0,Y 538.315,Z 268.278,A -85,B 0,C 180,E1 -4064.775,E2 -4064.775} C_VEL
LIN {X 0,Y 538.615,Z 245.676,A -85,B 0,C 180,E1 -4067.725,E2 -4067.725} C_VEL
LIN {X 0,Y 538.98,Z 222.272,A -85,B 0,C 180,E1 -4070.813,E2 -4070.813} C_VEL
LIN {X 0,Y 539.234,Z 199.625,A -85,B 0,C 180,E1 -4073.83,E2 -4073.83} C_VEL
LIN {X 0,Y 539.119,Z 193.51,A -85,B 0,C 180,E1 -4074.655,E2 -4074.655} C_VEL
LIN {X 0,Y 538.046,Z 187.466,A -85,B 0,C 180,E1 -4075.534,E2 -4075.534} C_VEL
LIN {X 0,Y 537.992,Z 187.468,A -85,B 0,C 180,E1 -4078.052,E2 -4078.052} C_VEL
LIN {X 0,Y 538.002,Z 187.471,A -85,B 0,C 180,E1 -4080.628,E2 -4080.628} C_VEL
LIN {X 0,Y 538.02,Z 187.467,A -85,B 0,C 180,E1 -4083.278,E2 -4083.278} C_VEL
LIN {X 0,Y 537.99,Z 187.466,A -85,B 0,C 180,E1 -4086.005,E2 -4086.005} C_VEL
LIN {X 0,Y 538.009,Z 187.471,A -85,B 0,C 180,E1 -4088.831,E2 -4088.831} C_VEL
LIN {X 0,Y 538.015,Z 187.463,A -85,B 0,C 180,E1 -4091.877,E2 -4091.877} C_VEL
LIN {X 0,Y 537.998,Z 187.47,A -85,B 0,C 180,E1 -4094.863,E2 -4094.863} C_VEL
LIN {X 0,Y 537.999,Z 187.465,A -85,B 0,C 180,E1 -4097.212,E2 -4097.212} C_VEL
LIN {X 0,Y 538.01,Z 187.468,A -85,B 0,C 180,E1 -4100.202,E2 -4100.202} C_VEL
LIN {X 0,Y 538.019,Z 187.464,A -85,B 0,C 180,E1 -4103.066,E2 -4103.066} C_VEL
LIN {X 0,Y 538.017,Z 187.464,A -85,B 0,C 180,E1 -4105.826,E2 -4105.826} C_VEL
LIN {X 0,Y 538.008,Z 187.469,A -85,B 0,C 180,E1 -4108.498,E2 -4108.498} C_VEL
LIN {X 0,Y 538.018,Z 187.462,A -85,B 0,C 180,E1 -4111.097,E2 -4111.097} C_VEL
LIN {X 0,Y 538.029,Z 187.463,A -85,B 0,C 180,E1 -4113.633,E2 -4113.633} C_VEL
LIN {X 0,Y 538.01,Z 187.463,A -85,B 0,C 180,E1 -4116.928,E2 -4116.928} C_VEL
LIN {X 0,Y 538.081,Z 187.46,A -85,B 0,C 180,E1 -4120.148,E2 -4120.148} C_VEL
LIN {X 0,Y 537.996,Z 187.466,A -85,B 0,C 180,E1 -4123.298,E2 -4123.298} C_VEL
LIN {X 0,Y 538.052,Z 187.465,A -85,B 0,C 180,E1 -4125.63,E2 -4125.63} C_VEL
LIN {X 0,Y 538.078,Z 187.454,A -85,B 0,C 180,E1 -4128.701,E2 -4128.701} C_VEL
LIN {X 0,Y 538.082,Z 187.462,A -85,B 0,C 180,E1 -4131.739,E2 -4131.739} C_VEL
LIN {X 0,Y 538.161,Z 187.445,A -85,B 0,C 180,E1 -4134.755,E2 -4134.755} C_VEL
LIN {X 0,Y 538.171,Z 187.447,A -85,B 0,C 180,E1 -4137.755,E2 -4137.755} C_VEL
LIN {X 0,Y 538.179,Z 187.444,A -85,B 0,C 180,E1 -4140.748,E2 -4140.748} C_VEL
LIN {X 0,Y 538.135,Z 187.454,A -85,B 0,C 180,E1 -4142.994,E2 -4142.994} C_VEL
LIN {X 0,Y 538.121,Z 187.45,A -85,B 0,C 180,E1 -4145.997,E2 -4145.997} C_VEL
LIN {X 0,Y 538.055,Z 187.466,A -85,B 0,C 180,E1 -4149.018,E2 -4149.018} C_VEL
LIN {X 0,Y 538.084,Z 187.456,A -85,B 0,C 180,E1 -4152.062,E2 -4152.062} C_VEL
LIN {X 0,Y 538.046,Z 187.467,A -85,B 0,C 180,E1 -4155.144,E2 -4155.144} C_VEL
LIN {X 0,Y 538.024,Z 187.465,A -85,B 0,C 180,E1 -4158.27,E2 -4158.27} C_VEL
LIN {X 0,Y 538.038,Z 187.468,A -85,B 0,C 180,E1 -4160.651,E2 -4160.651} C_VEL
LIN {X 0,Y 538.087,Z 187.647,A -85,B 0,C 180,E1 -4162.021,E2 -4162.021} C_VEL
LIN {X 0,Y 538.189,Z 194.627,A -85,B 0,C 180,E1 -4163.318,E2 -4163.318} C_VEL
LIN {X 0,Y 539.691,Z 202.962,A -85,B 0,C 180,E1 -4163.478,E2 -4163.478} C_VEL
LIN {X 0,Y 539.312,Z 301.264,A -85,B 0,C 180,E1 -4164.825,E2 -4164.825} C_VEL
LIN {X 0,Y 539.153,Z 314.634,A -85,B 0,C 180,E1 -4165.168,E2 -4165.168} C_VEL
LIN {X 0,Y 538.981,Z 327.545,A -85,B 0,C 180,E1 -4165.663,E2 -4165.663} C_VEL
LIN {X 0,Y 538.737,Z 340.157,A -85,B 0,C 180,E1 -4166.33,E2 -4166.33} C_VEL
LIN {X 0,Y 538.668,Z 344.054,A -85,B 0,C 180,E1 -4166.576,E2 -4166.576} C_VEL
LIN {X 0,Y 537.938,Z 349.092,A -85,B 0,C 180,E1 -4166.908,E2 -4166.908} C_VEL
LIN {X 0,Y 534.95,Z 356.999,A -85,B 0,C 180,E1 -4167.463,E2 -4167.463} C_VEL
LIN {X 0,Y 531.935,Z 364.418,A -85,B 0,C 180,E1 -4168.086,E2 -4168.086} C_VEL
LIN {X 0,Y 531.164,Z 368.633,A -85,B 0,C 180,E1 -4168.518,E2 -4168.518} C_VEL
LIN {X 0,Y 530.95,Z 376.975,A -85,B 0,C 180,E1 -4169.542,E2 -4169.542} C_VEL
LIN {X 0,Y 530.78,Z 385.246,A -85,B 0,C 180,E1 -4170.821,E2 -4170.821} C_VEL
LIN {X 0,Y 530.693,Z 391.532,A -85,B 0,C 180,E1 -4172.053,E2 -4172.053} C_VEL
LIN {X 0,Y 530.562,Z 396.879,A -85,B 0,C 180,E1 -4173.434,E2 -4173.434} C_VEL
LIN {X 0,Y 530.473,Z 400.594,A -85,B 0,C 180,E1 -4174.774,E2 -4174.774} C_VEL
LIN {X 0,Y 530.407,Z 402.94,A -85,B 0,C 180,E1 -4176.074,E2 -4176.074} C_VEL
LIN {X 0,Y 530.384,Z 404.172,A -85,B 0,C 180,E1 -4177.556,E2 -4177.556} C_VEL
LIN {X 0,Y 530.387,Z 404.155,A -85,B 0,C 180,E1 -4178.575,E2 -4178.575} C_VEL
LIN {X 0,Y 530.421,Z 403.213,A -85,B 0,C 180,E1 -4179.782,E2 -4179.782} C_VEL
LIN {X 0,Y 530.456,Z 401.325,A -85,B 0,C 180,E1 -4180.958,E2 -4180.958} C_VEL
LIN {X 0,Y 530.549,Z 397.321,A -85,B 0,C 180,E1 -4182.499,E2 -4182.499} C_VEL
LIN {X 0,Y 530.601,Z 393.603,A -85,B 0,C 180,E1 -4183.532,E2 -4183.532} C_VEL
LIN {X 0,Y 530.704,Z 387.767,A -85,B 0,C 180,E1 -4184.791,E2 -4184.791} C_VEL
LIN {X 0,Y 530.891,Z 380.152,A -85,B 0,C 180,E1 -4186.076,E2 -4186.076} C_VEL
LIN {X 0,Y 531.073,Z 372.189,A -85,B 0,C 180,E1 -4187.143,E2 -4187.143} C_VEL
LIN {X 0,Y 531.302,Z 362.318,A -85,B 0,C 180,E1 -4188.214,E2 -4188.214} C_VEL
LIN {X 0,Y 531.557,Z 351.916,A -85,B 0,C 180,E1 -4189.121,E2 -4189.121} C_VEL
LIN {X 0,Y 531.781,Z 341.103,A -85,B 0,C 180,E1 -4189.872,E2 -4189.872} C_VEL
LIN {X 0,Y 532.064,Z 328.79,A -85,B 0,C 180,E1 -4190.54,E2 -4190.54} C_VEL
LIN {X 0,Y 532.254,Z 316.219,A -85,B 0,C 180,E1 -4191.046,E2 -4191.046} C_VEL
LIN {X 0,Y 532.376,Z 303.337,A -85,B 0,C 180,E1 -4191.398,E2 -4191.398} C_VEL
LIN {X 0,Y 532.504,Z 281.14,A -85,B 0,C 180,E1 -4191.737,E2 -4191.737} C_VEL
LIN {X 0,Y 532.832,Z 203.723,A -85,B 0,C 180,E1 -4192.795,E2 -4192.795} C_VEL
LIN {X 0,Y 531.168,Z 194.81,A -85,B 0,C 180,E1 -4192.985,E2 -4192.985} C_VEL
LIN {X 0,Y 531.015,Z 188.34,A -85,B 0,C 180,E1 -4194.31,E2 -4194.31} C_VEL
LIN {X 0,Y 530.966,Z 188.349,A -85,B 0,C 180,E1 -4197.134,E2 -4197.134} C_VEL
LIN {X 0,Y 530.961,Z 188.343,A -85,B 0,C 180,E1 -4199.803,E2 -4199.803} C_VEL
LIN {X 0,Y 531.005,Z 188.336,A -85,B 0,C 180,E1 -4202.47,E2 -4202.47} C_VEL
LIN {X 0,Y 530.957,Z 188.348,A -85,B 0,C 180,E1 -4204.94,E2 -4204.94} C_VEL
LIN {X 0,Y 530.977,Z 188.339,A -85,B 0,C 180,E1 -4207.899,E2 -4207.899} C_VEL
LIN {X 0,Y 530.984,Z 188.343,A -85,B 0,C 180,E1 -4210.677,E2 -4210.677} C_VEL
LIN {X 0,Y 530.965,Z 188.347,A -85,B 0,C 180,E1 -4213.07,E2 -4213.07} C_VEL
LIN {X 0,Y 531.015,Z 188.336,A -85,B 0,C 180,E1 -4215.436,E2 -4215.436} C_VEL
LIN {X 0,Y 531.036,Z 188.337,A -85,B 0,C 180,E1 -4218.55,E2 -4218.55} C_VEL
LIN {X 0,Y 531.037,Z 188.332,A -85,B 0,C 180,E1 -4221.629,E2 -4221.629} C_VEL
LIN {X 0,Y 531.117,Z 188.33,A -85,B 0,C 180,E1 -4224.685,E2 -4224.685} C_VEL
LIN {X 0,Y 531.14,Z 188.319,A -85,B 0,C 180,E1 -4227.725,E2 -4227.725} C_VEL
LIN {X 0,Y 531.151,Z 188.322,A -85,B 0,C 180,E1 -4230.758,E2 -4230.758} C_VEL
LIN {X 0,Y 531.092,Z 188.326,A -85,B 0,C 180,E1 -4233.034,E2 -4233.034} C_VEL
LIN {X 0,Y 531.071,Z 188.332,A -85,B 0,C 180,E1 -4236.077,E2 -4236.077} C_VEL
LIN {X 0,Y 531.019,Z 188.334,A -85,B 0,C 180,E1 -4239.139,E2 -4239.139} C_VEL
LIN {X 0,Y 531.052,Z 188.332,A -85,B 0,C 180,E1 -4241.671,E2 -4241.671} C_VEL
LIN {X 0,Y 531.025,Z 188.333,A -85,B 0,C 180,E1 -4244.952,E2 -4244.952} C_VEL
LIN {X 0,Y 530.982,Z 188.342,A -85,B 0,C 180,E1 -4247.724,E2 -4247.724} C_VEL
LIN {X 0,Y 531.027,Z 188.34,A -85,B 0,C 180,E1 -4250.127,E2 -4250.127} C_VEL
LIN {X 0,Y 530.945,Z 188.344,A -85,B 0,C 180,E1 -4252.574,E2 -4252.574} C_VEL
LIN {X 0,Y 530.958,Z 188.342,A -85,B 0,C 180,E1 -4255.06,E2 -4255.06} C_VEL
LIN {X 0,Y 530.967,Z 188.346,A -85,B 0,C 180,E1 -4257.598,E2 -4257.598} C_VEL
LIN {X 0,Y 530.955,Z 188.345,A -85,B 0,C 180,E1 -4260.198,E2 -4260.198} C_VEL
LIN {X 0,Y 530.969,Z 188.34,A -85,B 0,C 180,E1 -4262.867,E2 -4262.867} C_VEL
LIN {X 0,Y 530.952,Z 188.351,A -85,B 0,C 180,E1 -4265.621,E2 -4265.621} C_VEL
LIN {X 0,Y 530.965,Z 188.341,A -85,B 0,C 180,E1 -4268.653,E2 -4268.653} C_VEL
LIN {X 0,Y 530.981,Z 188.347,A -85,B 0,C 180,E1 -4271.437,E2 -4271.437} C_VEL
LIN {X 0,Y 530.973,Z 188.34,A -85,B 0,C 180,E1 -4274.549,E2 -4274.549} C_VEL
LIN {X 0,Y 530.969,Z 188.343,A -85,B 0,C 180,E1 -4277.836,E2 -4277.836} C_VEL
LIN {X 0,Y 530.972,Z 188.34,A -85,B 0,C 180,E1 -4280.555,E2 -4280.555} C_VEL
LIN {X 0,Y 530.953,Z 188.348,A -85,B 0,C 180,E1 -4283.441,E2 -4283.441} C_VEL
LIN {X 0,Y 530.958,Z 188.341,A -85,B 0,C 180,E1 -4286.225,E2 -4286.225} C_VEL
LIN {X 0,Y 530.954,Z 188.348,A -85,B 0,C 180,E1 -4288.921,E2 -4288.921} C_VEL
LIN {X 0,Y 530.959,Z 188.344,A -85,B 0,C 180,E1 -4291.542,E2 -4291.542} C_VEL
LIN {X 0,Y 530.974,Z 188.34,A -85,B 0,C 180,E1 -4294.166,E2 -4294.166} C_VEL
LIN {X 0,Y 530.952,Z 188.347,A -85,B 0,C 180,E1 -4296.603,E2 -4296.603} C_VEL
LIN {X 0,Y 531.001,Z 188.342,A -85,B 0,C 180,E1 -4299.062,E2 -4299.062} C_VEL
LIN {X 0,Y 530.974,Z 188.34,A -85,B 0,C 180,E1 -4301.478,E2 -4301.478} C_VEL
LIN {X 0,Y 530.987,Z 188.346,A -85,B 0,C 180,E1 -4304.65,E2 -4304.65} C_VEL
LIN {X 0,Y 531.025,Z 188.333,A -85,B 0,C 180,E1 -4307.775,E2 -4307.775} C_VEL
LIN {X 0,Y 530.979,Z 188.341,A -85,B 0,C 180,E1 -4310.092,E2 -4310.092} C_VEL
LIN {X 0,Y 531.014,Z 188.341,A -85,B 0,C 180,E1 -4312.395,E2 -4312.395} C_VEL
LIN {X 0,Y 531.106,Z 188.329,A -85,B 0,C 180,E1 -4314.685,E2 -4314.685} C_VEL
LIN {X 0,Y 531.139,Z 188.32,A -85,B 0,C 180,E1 -4317.725,E2 -4317.725} C_VEL
LIN {X 0,Y 531.149,Z 188.321,A -85,B 0,C 180,E1 -4320.758,E2 -4320.758} C_VEL
LIN {X 0,Y 531.062,Z 188.329,A -85,B 0,C 180,E1 -4323.034,E2 -4323.034} C_VEL
LIN {X 0,Y 531.047,Z 188.337,A -85,B 0,C 180,E1 -4326.078,E2 -4326.078} C_VEL
LIN {X 0,Y 531.013,Z 188.335,A -85,B 0,C 180,E1 -4329.139,E2 -4329.139} C_VEL
LIN {X 0,Y 531.053,Z 188.333,A -85,B 0,C 180,E1 -4331.67,E2 -4331.67} C_VEL
LIN {X 0,Y 531.027,Z 188.333,A -85,B 0,C 180,E1 -4334.952,E2 -4334.952} C_VEL
LIN {X 0,Y 530.974,Z 188.345,A -85,B 0,C 180,E1 -4337.724,E2 -4337.724} C_VEL
LIN {X 0,Y 531.017,Z 188.34,A -85,B 0,C 180,E1 -4340.128,E2 -4340.128} C_VEL
LIN {X 0,Y 530.944,Z 188.344,A -85,B 0,C 180,E1 -4342.574,E2 -4342.574} C_VEL
LIN {X 0,Y 530.952,Z 188.343,A -85,B 0,C 180,E1 -4345.06,E2 -4345.06} C_VEL
LIN {X 0,Y 530.962,Z 188.348,A -85,B 0,C 180,E1 -4347.599,E2 -4347.599} C_VEL
LIN {X 0,Y 530.964,Z 188.341,A -85,B 0,C 180,E1 -4350.642,E2 -4350.642} C_VEL
LIN {X 0,Y 530.963,Z 188.349,A -85,B 0,C 180,E1 -4353.499,E2 -4353.499} C_VEL
LIN {X 0,Y 530.952,Z 188.342,A -85,B 0,C 180,E1 -4356.559,E2 -4356.559} C_VEL
LIN {X 0,Y 530.985,Z 188.347,A -85,B 0,C 180,E1 -4359.444,E2 -4359.444} C_VEL
LIN {X 0,Y 530.921,Z 188.346,A -85,B 0,C 180,E1 -4362.463,E2 -4362.463} C_VEL
LIN {X 0,Y 530.966,Z 188.347,A -85,B 0,C 180,E1 -4365.45,E2 -4365.45} C_VEL
LIN {X 0,Y 530.961,Z 188.342,A -85,B 0,C 180,E1 -4368.561,E2 -4368.561} C_VEL
LIN {X 0,Y 530.954,Z 188.345,A -85,B 0,C 180,E1 -4371.529,E2 -4371.529} C_VEL
LIN {X 0,Y 530.949,Z 188.343,A -85,B 0,C 180,E1 -4374.379,E2 -4374.379} C_VEL
LIN {X 0,Y 530.967,Z 188.348,A -85,B 0,C 180,E1 -4377.133,E2 -4377.133} C_VEL
LIN {X 0,Y 530.949,Z 188.344,A -85,B 0,C 180,E1 -4379.801,E2 -4379.801} C_VEL
LIN {X 0,Y 530.965,Z 188.347,A -85,B 0,C 180,E1 -4382.478,E2 -4382.478} C_VEL
LIN {X 0,Y 530.985,Z 188.377,A -85,B 0,C 180,E1 -4383.996,E2 -4383.996} C_VEL
LIN {X 0,Y 532.641,Z 197.398,A -85,B 0,C 180,E1 -4385.349,E2 -4385.349} C_VEL
LIN {X 0,Y 532.257,Z 215.736,A -85,B 0,C 180,E1 -4387.911,E2 -4387.911} C_VEL
LIN {X 0,Y 531.87,Z 237.709,A -85,B 0,C 180,E1 -4390.911,E2 -4390.911} C_VEL
LIN {X 0,Y 531.457,Z 259.639,A -85,B 0,C 180,E1 -4393.877,E2 -4393.877} C_VEL
LIN {X 0,Y 531.33,Z 268.258,A -85,B 0,C 180,E1 -4395.037,E2 -4395.037} C_VEL
LIN {X 0,Y 532.765,Z 280.013,A -85,B 0,C 180,E1 -4395.249,E2 -4395.249} C_VEL
LIN {X 0,Y 532.334,Z 377.59,A -85,B 0,C 180,E1 -4396.593,E2 -4396.593} C_VEL
LIN {X 0,Y 532.134,Z 390.822,A -85,B 0,C 180,E1 -4396.928,E2 -4396.928} C_VEL
LIN {X 0,Y 531.917,Z 403.559,A -85,B 0,C 180,E1 -4397.408,E2 -4397.408} C_VEL
LIN {X 0,Y 531.63,Z 415.716,A -85,B 0,C 180,E1 -4398.032,E2 -4398.032} C_VEL
LIN {X 0,Y 531.375,Z 427.927,A -85,B 0,C 180,E1 -4398.847,E2 -4398.847} C_VEL
LIN {X 0,Y 531.139,Z 438.246,A -85,B 0,C 180,E1 -4399.71,E2 -4399.71} C_VEL
LIN {X 0,Y 530.948,Z 447.524,A -85,B 0,C 180,E1 -4400.668,E2 -4400.668} C_VEL
LIN {X 0,Y 530.757,Z 456.558,A -85,B 0,C 180,E1 -4401.816,E2 -4401.816} C_VEL
LIN {X 0,Y 530.627,Z 463.836,A -85,B 0,C 180,E1 -4402.963,E2 -4402.963} C_VEL
LIN {X 0,Y 530.572,Z 470.468,A -85,B 0,C 180,E1 -4404.298,E2 -4404.298} C_VEL
LIN {X 0,Y 530.457,Z 474.848,A -85,B 0,C 180,E1 -4405.44,E2 -4405.44} C_VEL
LIN {X 0,Y 530.516,Z 477.174,A -85,B 0,C 180,E1 -4406.202,E2 -4406.202} C_VEL
LIN {X 0,Y 530.486,Z 479.054,A -85,B 0,C 180,E1 -4406.962,E2 -4406.962} C_VEL
LIN {X 0,Y 530.411,Z 480.461,A -85,B 0,C 180,E1 -4407.722,E2 -4407.722} C_VEL
LIN {X 0,Y 530.362,Z 482.077,A -85,B 0,C 180,E1 -4409.241,E2 -4409.241} C_VEL
LIN {X 0,Y 530.364,Z 482.293,A -85,B 0,C 180,E1 -4410,E2 -4410} C_VEL
LIN {X 0,Y 530.363,Z 482.072,A -85,B 0,C 180,E1 -4410.759,E2 -4410.759} C_VEL
LIN {X 0,Y 530.411,Z 480.45,A -85,B 0,C 180,E1 -4412.278,E2 -4412.278} C_VEL
LIN {X 0,Y 530.486,Z 479.037,A -85,B 0,C 180,E1 -4413.037,E2 -4413.037} C_VEL
LIN {X 0,Y 530.522,Z 476.063,A -85,B 0,C 180,E1 -4414.178,E2 -4414.178} C_VEL
LIN {X 0,Y 530.521,Z 472.033,A -85,B 0,C 180,E1 -4415.321,E2 -4415.321} C_VEL
LIN {X 0,Y 530.558,Z 466.436,A -85,B 0,C 180,E1 -4416.544,E2 -4416.544} C_VEL
LIN {X 0,Y 530.71,Z 459.073,A -85,B 0,C 180,E1 -4417.801,E2 -4417.801} C_VEL
LIN {X 0,Y 530.874,Z 450.677,A -85,B 0,C 180,E1 -4418.949,E2 -4418.949} C_VEL
LIN {X 0,Y 531.031,Z 442.063,A -85,B 0,C 180,E1 -4419.907,E2 -4419.907} C_VEL
LIN {X 0,Y 531.308,Z 431.436,A -85,B 0,C 180,E1 -4420.865,E2 -4420.865} C_VEL
LIN {X 0,Y 531.502,Z 420.706,A -85,B 0,C 180,E1 -4421.647,E2 -4421.647} C_VEL
LIN {X 0,Y 531.803,Z 409.373,A -85,B 0,C 180,E1 -4422.304,E2 -4422.304} C_VEL
LIN {X 0,Y 532.032,Z 397.451,A -85,B 0,C 180,E1 -4422.832,E2 -4422.832} C_VEL
LIN {X 0,Y 532.216,Z 383.704,A -85,B 0,C 180,E1 -4423.264,E2 -4423.264} C_VEL
LIN {X 0,Y 532.387,Z 371.392,A -85,B 0,C 180,E1 -4423.503,E2 -4423.503} C_VEL
LIN {X 0,Y 532.646,Z 278.22,A -85,B 0,C 180,E1 -4424.774,E2 -4424.774} C_VEL
LIN {X 0,Y 531.293,Z 267.737,A -85,B 0,C 180,E1 -4424.967,E2 -4424.967} C_VEL
LIN {X 0,Y 531.645,Z 243.965,A -85,B 0,C 180,E1 -4428.114,E2 -4428.114} C_VEL
LIN {X 0,Y 532.002,Z 221.639,A -85,B 0,C 180,E1 -4431.099,E2 -4431.099} C_VEL
LIN {X 0,Y 532.295,Z 198.924,A -85,B 0,C 180,E1 -4434.161,E2 -4434.161} C_VEL
LIN {X 0,Y 532.084,Z 194.168,A -85,B 0,C 180,E1 -4434.817,E2 -4434.817} C_VEL
LIN {X 0,Y 530.983,Z 188.345,A -85,B 0,C 180,E1 -4435.656,E2 -4435.656} C_VEL
LIN {X 0,Y 530.948,Z 188.348,A -85,B 0,C 180,E1 -4438.458,E2 -4438.458} C_VEL
LIN {X 0,Y 530.944,Z 188.352,A -85,B 0,C 180,E1 -4441.08,E2 -4441.08} C_VEL
LIN {X 0,Y 530.956,Z 188.343,A -85,B 0,C 180,E1 -4443.775,E2 -4443.775} C_VEL
LIN {X 0,Y 530.951,Z 188.348,A -85,B 0,C 180,E1 -4446.559,E2 -4446.559} C_VEL
LIN {X 0,Y 530.969,Z 188.342,A -85,B 0,C 180,E1 -4449.445,E2 -4449.445} C_VEL
LIN {X 0,Y 530.957,Z 188.348,A -85,B 0,C 180,E1 -4452.459,E2 -4452.459} C_VEL
LIN {X 0,Y 530.975,Z 188.339,A -85,B 0,C 180,E1 -4455.622,E2 -4455.622} C_VEL
LIN {X 0,Y 530.979,Z 188.347,A -85,B 0,C 180,E1 -4458.563,E2 -4458.563} C_VEL
LIN {X 0,Y 530.953,Z 188.343,A -85,B 0,C 180,E1 -4461.529,E2 -4461.529} C_VEL
LIN {X 0,Y 530.95,Z 188.35,A -85,B 0,C 180,E1 -4464.379,E2 -4464.379} C_VEL
LIN {X 0,Y 530.967,Z 188.34,A -85,B 0,C 180,E1 -4467.133,E2 -4467.133} C_VEL
LIN {X 0,Y 530.958,Z 188.346,A -85,B 0,C 180,E1 -4469.802,E2 -4469.802} C_VEL
LIN {X 0,Y 530.975,Z 188.343,A -85,B 0,C 180,E1 -4472.475,E2 -4472.475} C_VEL
LIN {X 0,Y 530.961,Z 188.342,A -85,B 0,C 180,E1 -4474.94,E2 -4474.94} C_VEL
LIN {X 0,Y 530.977,Z 188.347,A -85,B 0,C 180,E1 -4477.898,E2 -4477.898} C_VEL
LIN {X 0,Y 530.982,Z 188.34,A -85,B 0,C 180,E1 -4480.677,E2 -4480.677} C_VEL
LIN {X 0,Y 530.96,Z 188.341,A -85,B 0,C 180,E1 -4483.07,E2 -4483.07} C_VEL
LIN {X 0,Y 531.009,Z 188.339,A -85,B 0,C 180,E1 -4485.435,E2 -4485.435} C_VEL
LIN {X 0,Y 531.036,Z 188.331,A -85,B 0,C 180,E1 -4488.55,E2 -4488.55} C_VEL
LIN {X 0,Y 531.052,Z 188.338,A -85,B 0,C 180,E1 -4491.629,E2 -4491.629} C_VEL
LIN {X 0,Y 531.12,Z 188.322,A -85,B 0,C 180,E1 -4494.685,E2 -4494.685} C_VEL
LIN {X 0,Y 531.142,Z 188.323,A -85,B 0,C 180,E1 -4497.725,E2 -4497.725} C_VEL
LIN {X 0,Y 531.15,Z 188.32,A -85,B 0,C 180,E1 -4500.758,E2 -4500.758} C_VEL
LIN {X 0,Y 531.102,Z 188.33,A -85,B 0,C 180,E1 -4503.034,E2 -4503.034} C_VEL
LIN {X 0,Y 531.075,Z 188.328,A -85,B 0,C 180,E1 -4506.077,E2 -4506.077} C_VEL
LIN {X 0,Y 531.017,Z 188.343,A -85,B 0,C 180,E1 -4509.138,E2 -4509.138} C_VEL
LIN {X 0,Y 531.041,Z 188.334,A -85,B 0,C 180,E1 -4512.225,E2 -4512.225} C_VEL
LIN {X 0,Y 530.996,Z 188.343,A -85,B 0,C 180,E1 -4515.35,E2 -4515.35} C_VEL
LIN {X 0,Y 530.985,Z 188.345,A -85,B 0,C 180,E1 -4518.521,E2 -4518.521} C_VEL
LIN {X 0,Y 531.005,Z 188.345,A -85,B 0,C 180,E1 -4520.938,E2 -4520.938} C_VEL
LIN {X 0,Y 531.038,Z 188.372,A -85,B 0,C 180,E1 -4521.892,E2 -4521.892} C_VEL
LIN {X 0,Y 531.198,Z 194.855,A -85,B 0,C 180,E1 -4523.102,E2 -4523.102} C_VEL
LIN {X 0,Y 532.834,Z 203.288,A -85,B 0,C 180,E1 -4523.284,E2 -4523.284} C_VEL
LIN {X 0,Y 532.393,Z 301.859,A -85,B 0,C 180,E1 -4524.658,E2 -4524.658} C_VEL
LIN {X 0,Y 532.242,Z 314.875,A -85,B 0,C 180,E1 -4524.995,E2 -4524.995} C_VEL
LIN {X 0,Y 532.085,Z 327.359,A -85,B 0,C 180,E1 -4525.474,E2 -4525.474} C_VEL
LIN {X 0,Y 531.835,Z 339.657,A -85,B 0,C 180,E1 -4526.119,E2 -4526.119} C_VEL
LIN {X 0,Y 531.558,Z 351.517,A -85,B 0,C 180,E1 -4526.926,E2 -4526.926} C_VEL
LIN {X 0,Y 531.34,Z 361.391,A -85,B 0,C 180,E1 -4527.77,E2 -4527.77} C_VEL
LIN {X 0,Y 531.164,Z 368.633,A -85,B 0,C 180,E1 -4528.518,E2 -4528.518} C_VEL
LIN {X 0,Y 530.4,Z 372.705,A -85,B 0,C 180,E1 -4528.975,E2 -4528.975} C_VEL
LIN {X 0,Y 527.395,Z 379.001,A -85,B 0,C 180,E1 -4529.74,E2 -4529.74} C_VEL
LIN {X 0,Y 524.418,Z 384.743,A -85,B 0,C 180,E1 -4530.563,E2 -4530.563} C_VEL
LIN {X 0,Y 523.699,Z 387.83,A -85,B 0,C 180,E1 -4531.105,E2 -4531.105} C_VEL
LIN {X 0,Y 523.58,Z 393.269,A -85,B 0,C 180,E1 -4532.259,E2 -4532.259} C_VEL
LIN {X 0,Y 523.499,Z 398.309,A -85,B 0,C 180,E1 -4533.659,E2 -4533.659} C_VEL
LIN {X 0,Y 523.392,Z 401.731,A -85,B 0,C 180,E1 -4535.006,E2 -4535.006} C_VEL
LIN {X 0,Y 523.327,Z 403.797,A -85,B 0,C 180,E1 -4536.316,E2 -4536.316} C_VEL
LIN {X 0,Y 523.329,Z 404.702,A -85,B 0,C 180,E1 -4537.596,E2 -4537.596} C_VEL
LIN {X 0,Y 523.316,Z 404.361,A -85,B 0,C 180,E1 -4539.139,E2 -4539.139} C_VEL
LIN {X 0,Y 523.372,Z 403.293,A -85,B 0,C 180,E1 -4540.133,E2 -4540.133} C_VEL
LIN {X 0,Y 523.445,Z 400.332,A -85,B 0,C 180,E1 -4541.672,E2 -4541.672} C_VEL
LIN {X 0,Y 523.516,Z 397.133,A -85,B 0,C 180,E1 -4542.774,E2 -4542.774} C_VEL
LIN {X 0,Y 523.551,Z 392.99,A -85,B 0,C 180,E1 -4543.873,E2 -4543.873} C_VEL
LIN {X 0,Y 523.7,Z 386.848,A -85,B 0,C 180,E1 -4545.15,E2 -4545.15} C_VEL
LIN {X 0,Y 523.889,Z 378.995,A -85,B 0,C 180,E1 -4546.42,E2 -4546.42} C_VEL
LIN {X 0,Y 524.137,Z 370.54,A -85,B 0,C 180,E1 -4547.517,E2 -4547.517} C_VEL
LIN {X 0,Y 524.368,Z 361.182,A -85,B 0,C 180,E1 -4548.504,E2 -4548.504} C_VEL
LIN {X 0,Y 524.621,Z 350.581,A -85,B 0,C 180,E1 -4549.402,E2 -4549.402} C_VEL
LIN {X 0,Y 524.891,Z 339.948,A -85,B 0,C 180,E1 -4550.126,E2 -4550.126} C_VEL
LIN {X 0,Y 525.184,Z 328.464,A -85,B 0,C 180,E1 -4550.74,E2 -4550.74} C_VEL
LIN {X 0,Y 525.348,Z 315.839,A -85,B 0,C 180,E1 -4551.242,E2 -4551.242} C_VEL
LIN {X 0,Y 525.473,Z 302.216,A -85,B 0,C 180,E1 -4551.605,E2 -4551.605} C_VEL
LIN {X 0,Y 526.013,Z 204.611,A -85,B 0,C 180,E1 -4552.984,E2 -4552.984} C_VEL
LIN {X 0,Y 524.183,Z 195.161,A -85,B 0,C 180,E1 -4553.191,E2 -4553.191} C_VEL
LIN {X 0,Y 523.993,Z 189.261,A -85,B 0,C 180,E1 -4554.396,E2 -4554.396} C_VEL
LIN {X 0,Y 523.935,Z 189.221,A -85,B 0,C 180,E1 -4557.68,E2 -4557.68} C_VEL
LIN {X 0,Y 523.954,Z 189.216,A -85,B 0,C 180,E1 -4560.677,E2 -4560.677} C_VEL
LIN {X 0,Y 523.938,Z 189.221,A -85,B 0,C 180,E1 -4562.866,E2 -4562.866} C_VEL
LIN {X 0,Y 523.935,Z 189.217,A -85,B 0,C 180,E1 -4565.804,E2 -4565.804} C_VEL
LIN {X 0,Y 523.946,Z 189.22,A -85,B 0,C 180,E1 -4568.767,E2 -4568.767} C_VEL
LIN {X 0,Y 523.939,Z 189.221,A -85,B 0,C 180,E1 -4571.22,E2 -4571.22} C_VEL
LIN {X 0,Y 523.923,Z 189.218,A -85,B 0,C 180,E1 -4573.639,E2 -4573.639} C_VEL
LIN {X 0,Y 523.93,Z 189.217,A -85,B 0,C 180,E1 -4576.028,E2 -4576.028} C_VEL
LIN {X 0,Y 524.015,Z 189.21,A -85,B 0,C 180,E1 -4578.394,E2 -4578.394} C_VEL
LIN {X 0,Y 523.989,Z 189.21,A -85,B 0,C 180,E1 -4581.516,E2 -4581.516} C_VEL
LIN {X 0,Y 524.078,Z 189.208,A -85,B 0,C 180,E1 -4584.614,E2 -4584.614} C_VEL
LIN {X 0,Y 524.112,Z 189.194,A -85,B 0,C 180,E1 -4587.695,E2 -4587.695} C_VEL
LIN {X 0,Y 524.122,Z 189.198,A -85,B 0,C 180,E1 -4590.769,E2 -4590.769} C_VEL
LIN {X 0,Y 524.033,Z 189.205,A -85,B 0,C 180,E1 -4593.075,E2 -4593.075} C_VEL
LIN {X 0,Y 524.029,Z 189.211,A -85,B 0,C 180,E1 -4596.159,E2 -4596.159} C_VEL
LIN {X 0,Y 523.988,Z 189.21,A -85,B 0,C 180,E1 -4599.262,E2 -4599.262} C_VEL
LIN {X 0,Y 524.001,Z 189.21,A -85,B 0,C 180,E1 -4601.737,E2 -4601.737} C_VEL
LIN {X 0,Y 523.989,Z 189.21,A -85,B 0,C 180,E1 -4605.05,E2 -4605.05} C_VEL
LIN {X 0,Y 523.946,Z 189.222,A -85,B 0,C 180,E1 -4607.97,E2 -4607.97} C_VEL
LIN {X 0,Y 523.96,Z 189.217,A -85,B 0,C 180,E1 -4610.411,E2 -4610.411} C_VEL
LIN {X 0,Y 523.91,Z 189.219,A -85,B 0,C 180,E1 -4612.894,E2 -4612.894} C_VEL
LIN {X 0,Y 523.907,Z 189.222,A -85,B 0,C 180,E1 -4615.421,E2 -4615.421} C_VEL
LIN {X 0,Y 523.917,Z 189.225,A -85,B 0,C 180,E1 -4618.002,E2 -4618.002} C_VEL
LIN {X 0,Y 523.937,Z 189.216,A -85,B 0,C 180,E1 -4620.853,E2 -4620.853} C_VEL
LIN {X 0,Y 523.961,Z 189.222,A -85,B 0,C 180,E1 -4623.734,E2 -4623.734} C_VEL
LIN {X 0,Y 523.901,Z 189.221,A -85,B 0,C 180,E1 -4626.401,E2 -4626.401} C_VEL
LIN {X 0,Y 523.915,Z 189.221,A -85,B 0,C 180,E1 -4629.086,E2 -4629.086} C_VEL
LIN {X 0,Y 523.942,Z 189.217,A -85,B 0,C 180,E1 -4632.12,E2 -4632.12} C_VEL
LIN {X 0,Y 523.94,Z 189.223,A -85,B 0,C 180,E1 -4635.311,E2 -4635.311} C_VEL
LIN {X 0,Y 523.942,Z 189.217,A -85,B 0,C 180,E1 -4638.692,E2 -4638.692} C_VEL
LIN {X 0,Y 523.915,Z 189.22,A -85,B 0,C 180,E1 -4641.898,E2 -4641.898} C_VEL
LIN {X 0,Y 523.924,Z 189.222,A -85,B 0,C 180,E1 -4644.912,E2 -4644.912} C_VEL
LIN {X 0,Y 523.936,Z 189.218,A -85,B 0,C 180,E1 -4647.68,E2 -4647.68} C_VEL
LIN {X 0,Y 523.938,Z 189.219,A -85,B 0,C 180,E1 -4650.68,E2 -4650.68} C_VEL
LIN {X 0,Y 523.935,Z 189.217,A -85,B 0,C 180,E1 -4653.726,E2 -4653.726} C_VEL
LIN {X 0,Y 523.91,Z 189.22,A -85,B 0,C 180,E1 -4656.269,E2 -4656.269} C_VEL
LIN {X 0,Y 523.948,Z 189.222,A -85,B 0,C 180,E1 -4658.767,E2 -4658.767} C_VEL
LIN {X 0,Y 523.938,Z 189.219,A -85,B 0,C 180,E1 -4661.22,E2 -4661.22} C_VEL
LIN {X 0,Y 523.911,Z 189.219,A -85,B 0,C 180,E1 -4663.638,E2 -4663.638} C_VEL
LIN {X 0,Y 523.919,Z 189.219,A -85,B 0,C 180,E1 -4666.027,E2 -4666.027} C_VEL
LIN {X 0,Y 524.017,Z 189.211,A -85,B 0,C 180,E1 -4668.394,E2 -4668.394} C_VEL
LIN {X 0,Y 523.988,Z 189.21,A -85,B 0,C 180,E1 -4671.516,E2 -4671.516} C_VEL
LIN {X 0,Y 524.067,Z 189.207,A -85,B 0,C 180,E1 -4674.614,E2 -4674.614} C_VEL
LIN {X 0,Y 524.111,Z 189.195,A -85,B 0,C 180,E1 -4677.695,E2 -4677.695} C_VEL
LIN {X 0,Y 524.119,Z 189.196,A -85,B 0,C 180,E1 -4680.768,E2 -4680.768} C_VEL
LIN {X 0,Y 524.005,Z 189.208,A -85,B 0,C 180,E1 -4683.075,E2 -4683.075} C_VEL
LIN {X 0,Y 524.009,Z 189.215,A -85,B 0,C 180,E1 -4686.16,E2 -4686.16} C_VEL
LIN {X 0,Y 523.983,Z 189.21,A -85,B 0,C 180,E1 -4689.262,E2 -4689.262} C_VEL
LIN {X 0,Y 524.002,Z 189.212,A -85,B 0,C 180,E1 -4691.737,E2 -4691.737} C_VEL
LIN {X 0,Y 523.99,Z 189.209,A -85,B 0,C 180,E1 -4695.049,E2 -4695.049} C_VEL
LIN {X 0,Y 523.917,Z 189.227,A -85,B 0,C 180,E1 -4697.971,E2 -4697.971} C_VEL
LIN {X 0,Y 523.953,Z 189.216,A -85,B 0,C 180,E1 -4700.411,E2 -4700.411} C_VEL
LIN {X 0,Y 523.91,Z 189.219,A -85,B 0,C 180,E1 -4702.894,E2 -4702.894} C_VEL
LIN {X 0,Y 523.902,Z 189.224,A -85,B 0,C 180,E1 -4705.421,E2 -4705.421} C_VEL
LIN {X 0,Y 523.909,Z 189.224,A -85,B 0,C 180,E1 -4708.003,E2 -4708.003} C_VEL
LIN {X 0,Y 523.938,Z 189.216,A -85,B 0,C 180,E1 -4710.853,E2 -4710.853} C_VEL
LIN {X 0,Y 523.929,Z 189.224,A -85,B 0,C 180,E1 -4713.729,E2 -4713.729} C_VEL
LIN {X 0,Y 523.9,Z 189.221,A -85,B 0,C 180,E1 -4716.4,E2 -4716.4} C_VEL
LIN {X 0,Y 523.92,Z 189.222,A -85,B 0,C 180,E1 -4719.085,E2 -4719.085} C_VEL
LIN {X 0,Y 523.901,Z 189.221,A -85,B 0,C 180,E1 -4722.124,E2 -4722.124} C_VEL
LIN {X 0,Y 523.936,Z 189.225,A -85,B 0,C 180,E1 -4725.311,E2 -4725.311} C_VEL
LIN {X 0,Y 523.922,Z 189.22,A -85,B 0,C 180,E1 -4728.694,E2 -4728.694} C_VEL
LIN {X 0,Y 523.914,Z 189.219,A -85,B 0,C 180,E1 -4731.898,E2 -4731.898} C_VEL
LIN {X 0,Y 523.92,Z 189.225,A -85,B 0,C 180,E1 -4734.912,E2 -4734.912} C_VEL
LIN {X 0,Y 523.933,Z 189.219,A -85,B 0,C 180,E1 -4737.681,E2 -4737.681} C_VEL
LIN {X 0,Y 523.938,Z 189.223,A -85,B 0,C 180,E1 -4740.68,E2 -4740.68} C_VEL
LIN {X 0,Y 523.939,Z 189.243,A -85,B 0,C 180,E1 -4743.811,E2 -4743.811} C_VEL
LIN {X 0,Y 525.585,Z 197.488,A -85,B 0,C 180,E1 -4745.073,E2 -4745.073} C_VEL
LIN {X 0,Y 525.61,Z 204.954,A -85,B 0,C 180,E1 -4746.141,E2 -4746.141} C_VEL
LIN {X 0,Y 525.135,Z 225.633,A -85,B 0,C 180,E1 -4749.043,E2 -4749.043} C_VEL
LIN {X 0,Y 524.688,Z 247.483,A -85,B 0,C 180,E1 -4752.056,E2 -4752.056} C_VEL
LIN {X 0,Y 524.282,Z 267.78,A -85,B 0,C 180,E1 -4754.832,E2 -4754.832} C_VEL
LIN {X 0,Y 525.874,Z 281.029,A -85,B 0,C 180,E1 -4755.072,E2 -4755.072} C_VEL
LIN {X 0,Y 525.42,Z 376.814,A -85,B 0,C 180,E1 -4756.413,E2 -4756.413} C_VEL
LIN {X 0,Y 525.175,Z 390.131,A -85,B 0,C 180,E1 -4756.752,E2 -4756.752} C_VEL
LIN {X 0,Y 524.948,Z 402.914,A -85,B 0,C 180,E1 -4757.238,E2 -4757.238} C_VEL
LIN {X 0,Y 524.679,Z 414.352,A -85,B 0,C 180,E1 -4757.824,E2 -4757.824} C_VEL
LIN {X 0,Y 524.412,Z 426.041,A -85,B 0,C 180,E1 -4758.599,E2 -4758.599} C_VEL
LIN {X 0,Y 524.155,Z 436.613,A -85,B 0,C 180,E1 -4759.473,E2 -4759.473} C_VEL
LIN {X 0,Y 523.893,Z 445.257,A -85,B 0,C 180,E1 -4760.346,E2 -4760.346} C_VEL
LIN {X 0,Y 523.74,Z 453.239,A -85,B 0,C 180,E1 -4761.317,E2 -4761.317} C_VEL
LIN {X 0,Y 523.575,Z 461.038,A -85,B 0,C 180,E1 -4762.48,E2 -4762.48} C_VEL
LIN {X 0,Y 523.467,Z 468.218,A -85,B 0,C 180,E1 -4763.834,E2 -4763.834} C_VEL
LIN {X 0,Y 523.383,Z 472.996,A -85,B 0,C 180,E1 -4764.993,E2 -4764.993} C_VEL
LIN {X 0,Y 523.443,Z 476.655,A -85,B 0,C 180,E1 -4766.15,E2 -4766.15} C_VEL
LIN {X 0,Y 523.423,Z 478.537,A -85,B 0,C 180,E1 -4766.921,E2 -4766.921} C_VEL
LIN {X 0,Y 523.336,Z 479.944,A -85,B 0,C 180,E1 -4767.691,E2 -4767.691} C_VEL
LIN {X 0,Y 523.28,Z 481.558,A -85,B 0,C 180,E1 -4769.23,E2 -4769.23} C_VEL
LIN {X 0,Y 523.284,Z 481.772,A -85,B 0,C 180,E1 -4770,E2 -4770} C_VEL
LIN {X 0,Y 523.281,Z 481.55,A -85,B 0,C 180,E1 -4770.769,E2 -4770.769} C_VEL
LIN {X 0,Y 523.336,Z 479.921,A -85,B 0,C 180,E1 -4772.309,E2 -4772.309} C_VEL
LIN {X 0,Y 523.423,Z 478.504,A -85,B 0,C 180,E1 -4773.079,E2 -4773.079} C_VEL
LIN {X 0,Y 523.441,Z 475.52,A -85,B 0,C 180,E1 -4774.235,E2 -4774.235} C_VEL
LIN {X 0,Y 523.455,Z 471.48,A -85,B 0,C 180,E1 -4775.393,E2 -4775.393} C_VEL
LIN {X 0,Y 523.535,Z 465.315,A -85,B 0,C 180,E1 -4776.737,E2 -4776.737} C_VEL
LIN {X 0,Y 523.652,Z 458.493,A -85,B 0,C 180,E1 -4777.907,E2 -4777.907} C_VEL
LIN {X 0,Y 523.805,Z 450.076,A -85,B 0,C 180,E1 -4779.07,E2 -4779.07} C_VEL
LIN {X 0,Y 523.982,Z 441.442,A -85,B 0,C 180,E1 -4780.041,E2 -4780.041} C_VEL
LIN {X 0,Y 524.292,Z 430.794,A -85,B 0,C 180,E1 -4781.012,E2 -4781.012} C_VEL
LIN {X 0,Y 524.502,Z 419.418,A -85,B 0,C 180,E1 -4781.847,E2 -4781.847} C_VEL
LIN {X 0,Y 524.807,Z 408.668,A -85,B 0,C 180,E1 -4782.47,E2 -4782.47} C_VEL
LIN {X 0,Y 525.053,Z 396.687,A -85,B 0,C 180,E1 -4783.005,E2 -4783.005} C_VEL
LIN {X 0,Y 525.275,Z 382.869,A -85,B 0,C 180,E1 -4783.442,E2 -4783.442} C_VEL
LIN {X 0,Y 525.49,Z 370.348,A -85,B 0,C 180,E1 -4783.683,E2 -4783.683} C_VEL
LIN {X 0,Y 525.753,Z 278.47,A -85,B 0,C 180,E1 -4784.961,E2 -4784.961} C_VEL
LIN {X 0,Y 524.262,Z 267.109,A -85,B 0,C 180,E1 -4785.177,E2 -4785.177} C_VEL
LIN {X 0,Y 524.633,Z 243.774,A -85,B 0,C 180,E1 -4788.309,E2 -4788.309} C_VEL
LIN {X 0,Y 525.019,Z 222.504,A -85,B 0,C 180,E1 -4791.188,E2 -4791.188} C_VEL
LIN {X 0,Y 525.357,Z 199.76,A -85,B 0,C 180,E1 -4794.29,E2 -4794.29} C_VEL
LIN {X 0,Y 525.097,Z 195.142,A -85,B 0,C 180,E1 -4794.935,E2 -4794.935} C_VEL
LIN {X 0,Y 523.946,Z 189.221,A -85,B 0,C 180,E1 -4795.811,E2 -4795.811} C_VEL
LIN {X 0,Y 523.905,Z 189.23,A -85,B 0,C 180,E1 -4798.877,E2 -4798.877} C_VEL
LIN {X 0,Y 523.911,Z 189.223,A -85,B 0,C 180,E1 -4801.545,E2 -4801.545} C_VEL
LIN {X 0,Y 523.919,Z 189.221,A -85,B 0,C 180,E1 -4804.291,E2 -4804.291} C_VEL
LIN {X 0,Y 523.905,Z 189.226,A -85,B 0,C 180,E1 -4807.132,E2 -4807.132} C_VEL
LIN {X 0,Y 523.913,Z 189.221,A -85,B 0,C 180,E1 -4810.126,E2 -4810.126} C_VEL
LIN {X 0,Y 523.917,Z 189.225,A -85,B 0,C 180,E1 -4812.456,E2 -4812.456} C_VEL
LIN {X 0,Y 523.94,Z 189.216,A -85,B 0,C 180,E1 -4815.31,E2 -4815.31} C_VEL
LIN {X 0,Y 523.94,Z 189.222,A -85,B 0,C 180,E1 -4818.692,E2 -4818.692} C_VEL
LIN {X 0,Y 523.913,Z 189.222,A -85,B 0,C 180,E1 -4821.898,E2 -4821.898} C_VEL
LIN {X 0,Y 523.923,Z 189.219,A -85,B 0,C 180,E1 -4824.911,E2 -4824.911} C_VEL
LIN {X 0,Y 523.935,Z 189.218,A -85,B 0,C 180,E1 -4827.68,E2 -4827.68} C_VEL
LIN {X 0,Y 523.952,Z 189.216,A -85,B 0,C 180,E1 -4830.677,E2 -4830.677} C_VEL
LIN {X 0,Y 523.933,Z 189.22,A -85,B 0,C 180,E1 -4833.726,E2 -4833.726} C_VEL
LIN {X 0,Y 523.909,Z 189.225,A -85,B 0,C 180,E1 -4836.269,E2 -4836.269} C_VEL
LIN {X 0,Y 523.945,Z 189.215,A -85,B 0,C 180,E1 -4838.767,E2 -4838.767} C_VEL
LIN {X 0,Y 523.937,Z 189.218,A -85,B 0,C 180,E1 -4841.22,E2 -4841.22} C_VEL
LIN {X 0,Y 523.917,Z 189.224,A -85,B 0,C 180,E1 -4843.638,E2 -4843.638} C_VEL
LIN {X 0,Y 523.928,Z 189.222,A -85,B 0,C 180,E1 -4846.028,E2 -4846.028} C_VEL
LIN {X 0,Y 524.013,Z 189.207,A -85,B 0,C 180,E1 -4848.394,E2 -4848.394} C_VEL
LIN {X 0,Y 524,Z 189.215,A -85,B 0,C 180,E1 -4851.516,E2 -4851.516} C_VEL
LIN {X 0,Y 524.081,Z 189.199,A -85,B 0,C 180,E1 -4854.614,E2 -4854.614} C_VEL
LIN {X 0,Y 524.114,Z 189.199,A -85,B 0,C 180,E1 -4857.694,E2 -4857.694} C_VEL
LIN {X 0,Y 524.121,Z 189.196,A -85,B 0,C 180,E1 -4860.768,E2 -4860.768} C_VEL
LIN {X 0,Y 524.07,Z 189.207,A -85,B 0,C 180,E1 -4863.075,E2 -4863.075} C_VEL
LIN {X 0,Y 524.034,Z 189.205,A -85,B 0,C 180,E1 -4866.159,E2 -4866.159} C_VEL
LIN {X 0,Y 523.987,Z 189.218,A -85,B 0,C 180,E1 -4869.262,E2 -4869.262} C_VEL
LIN {X 0,Y 524.003,Z 189.212,A -85,B 0,C 180,E1 -4871.739,E2 -4871.739} C_VEL
LIN {X 0,Y 523.994,Z 189.219,A -85,B 0,C 180,E1 -4875.052,E2 -4875.052} C_VEL
LIN {X 0,Y 523.947,Z 189.217,A -85,B 0,C 180,E1 -4877.97,E2 -4877.97} C_VEL
LIN {X 0,Y 523.974,Z 189.218,A -85,B 0,C 180,E1 -4880.41,E2 -4880.41} C_VEL
LIN {X 0,Y 523.989,Z 189.338,A -85,B 0,C 180,E1 -4881.799,E2 -4881.799} C_VEL
